(* CODESYS project aspersao_v1_1_0.library
   Company: Teknike
   DefaultNamespace: Teknike_Aspersao
   Version: 1.1.0
   Placeholder: Teknike_Aspersao
   Author: Tiago B. Cunico
   Description: Biblioteca para controle de aspersao
   Title: Aspersao

Project tree, tasks and I/O mapping:
  libraries: OSCAT - AixOCAT, * (RWTH Aachen University - E.ON Energy Research Center); Tc2_ControllerToolbox, * (Beckhoff Automation GmbH); Tc2_Standard, * (Beckhoff Automation GmbH); Tc2_System, * (Beckhoff Automation GmbH); Tc2_TcpIp, * (Beckhoff Automation GmbH); Tc2_Utilities, * (Beckhoff Automation GmbH); Tc3_Database, * (Beckhoff Automation GmbH); Tc3_Module, * (Beckhoff Automation GmbH); Geral, * (Teknike); Partidas, * (Teknike); Sensores, * (Teknike); SQL, * (Teknike); TwinCAT Dynamic String Kit, * (FisoThemes)
  POUs/
    Automatico/
      Aspercao/
        Balanca/
          function block FB_Balanca [ST]
          function block FB_SalvaBalancaBanco [ST]
          data type st_Balanca
        Camaras/
          Cluster/
            data type st_Cluster
            data type st_Cluster_Entrada
            data type st_Cluster_Interno
            data type st_Cluster_Saida
          function block FB_Camaras [ST]: AjustaSaidaPeV, AtualizaValvulasDosClusters, ContrlCamaras, ContrlCluster, ContrlEntreClusters, SalvaAbreEFechaNoCluster, DefineQuandoSalvaEvento, EventosRelatorio, fimAspersao, FimResfriamento, GeraRelatorio, InicioAspercao, InicioResfriamento, SalvaGrafico, SalvaProtocolo, AjustaEntrada, AjustaSaida, ControleLed, InicioPelaCamara, Status
          function block FB_SalvaEventoRelatorio [ST]: SalvaEvento
          data type st_Camara
          data type st_Camara_Config
          data type st_camara_Entradas
          data type st_camara_Saidas
          data type st_Camara_Status
          data type st_EventoRelatorio
        ControleLiberacaoCamaras/
          AreaFria/
            Sts/
              data type st_AreaFria
              data type st_AreaFriaControle
              data type st_SupervisorioAreaFria
            function block FB_ControleSaidaAreaFria [ST]: DefineQuandoSalvaEvento, EscrevePesoFrioCarcaca, EscrevePesoFrioProcesso, FimRefrimento, GeraRelatorio, IgnoraCarcacaBanco, SalvaEvento, AjustaEntrada, AjustaSaida, PegaCamarasDisponiveis, VeCarcacasAIgnorar
          AreaQuente/
            Sts/
              data type st_AreaQuente
              data type st_AreaQuenteControle
              data type st_SupCamarasDisponiveis
              data type st_SupervisorioAreaQuente
            function block FB_ControleEntradaAreaQuente [ST]: Cancela, EscreveNovaCarcacaBanco, EscreveNovoProcessoBanco, EscrevePesoQuenteProcesso, AjustaEntrada, AjustaSaida, PegaCamarasDisponiveis
          Funcionamento_TODO.txt
          data type st_CarcacaBD
          data type st_ProcessoBD
        ControleProtocolo/
          function block FB_ControleEdicaoProtocolo [ST]
          data type st_DBProtocolo
          data type st_Protocolo
        ControleValvulas/
          function block FB_ControleValvulaApersao [ST]: AjustaBanco, ControleEventos, EventosRelatorio, HoraTermina, LogBanco, SalvaAbreEFecha, AjustaEntrada, AjustaSaida, CancelaProtocolo, TempoMaximoDeProtocolo, VSAr
          data type st_ConfigControleValvula
          data type st_ControleValvula
          data type st_enControleValvulas
          data type st_saControleValvulas
          data type st_ValvulasBD
        RFIDeBalanca/
          function block FB_RFIDBalancaChoque [ST]: ControlePeso, ControleTAG
          function block FB_RFIDBalancaEntrada [ST]: ControlePeso, ControleTAG
          function block FB_RFIDBalancaSaida [ST]: ControlePeso, ControleTAG
          data type st_BufferTagBalanca
          data type st_RFIDdb
          data type st_RFIDePeso
      ControlesPID/
        Estruturas/
          data type stConfigMaxMinSet
          data type stControlePID
          data type stPID
          data type stPID_EN
          data type stPID_SA
        function block FB_PIDeGrafico [ST]: aPID, Grafico, TextoErro, TextoStatus
        data type st_Anel
        data type st_Tanque
    Comunicacao/
      sts/
        areafria/
          data type st_EnIHMAreaFria
          data type st_IHMAreaFria
          data type st_SaIHMAreaFria
        areaquente/
          data type st_EnIHMAreaQuente
          data type st_IHMAreaQuente
          data type st_SaIHMAreaQuente
        CamaraLRV/
          data type st_CamaraLRV
          data type st_En_CamaraLRV
          data type st_Sa_CamaraLRV
          data type st_StatusCamaras
        Camaras/
          data type st_En_IHMCamaras
          data type st_IHMCamara
          data type st_Sa_IHMCamaras
    global variables GVL_BlibliotecaAspersao
    program MAIN [ST]
    program ValidaLicensa [ST]: Licensas
  00000000-0000-0000-0000-000000000000|POUs\Automatico\Aspercao\ControleLiberacaoCamaras\Funcionamento_TODO.txt
*)

// POUs/Automatico/Aspercao/Balanca/st_Balanca
TYPE st_Balanca :
STRUCT
	xConecta : BOOL;	
	ip : T_IPv4Addr;
	xNovoResultado : BOOL;
	rPeso : REAL;
	xOnline : BOOL; //
	xResetContador : BOOL;
	iContador : UDINT;
	stBuffer : ARRAY[0..9] OF REAL;
END_STRUCT
END_TYPE

// POUs/Automatico/Aspercao/Camaras/Cluster/st_Cluster
TYPE st_Cluster :
STRUCT
	En 	: st_Cluster_Entrada;
	Sa 	: st_Cluster_Saida;
	i	: st_Cluster_Interno;
END_STRUCT
END_TYPE

// POUs/Automatico/Aspercao/Camaras/Cluster/st_Cluster_Entrada
TYPE st_Cluster_Entrada :
STRUCT
	iValvulas : ARRAY[0..20] OF INT;//Quais valvulas estao nesse cluster
	xPausaCluster : BOOL;//sinal da camara para sincronizar o cluster
	iPosisaoCluster : INT;//Em qual posição esse cluster esta, começa em 0
	rTempoEntreValvulas : REAL;//segundos entre cada 1 das valvulas
	xHabilitaEvaporador : ARRAY[0..10] OF BOOL;//Quais evaporadores vao parar quando esse cluster pedir
END_STRUCT
END_TYPE

// POUs/Automatico/Aspercao/Camaras/Cluster/st_Cluster_Interno
TYPE st_Cluster_Interno :
STRUCT
	
	
	rtMasterAbriu : R_TRIG;
	xHEaMestre : BOOL;
	dthrInicioValMestre : DT;//momento em que a valvula mestre inicio, usa pra saber quando libera o cluster
	xIniciaSincronismo : BOOL;// quando tru ele fica contando o tempo para quando for a hora liberar a valvula
	lrTempoTotal : LREAL;//essa é a divisao de quando cada valvula pode entrar, (tempo OFF mais Tempo ON)
	lrTempoDeCadaBloco : LREAL;//essa é a divisao de quando cada valvula pode entrar, (tempo OFF mais Tempo ON)/Numero de clusters
	lrPosicaoDeEntrada : LREAL;//momento em que a valvula pode entrar mesmo
	
	iEtapaAnterior : INT;
	
	rtIniciaSincronismo : R_TRIG;
	rtTrocouEtapa : R_TRIG;
	
	tonSincornismo : TON_P;
	TonMomentoDeEntrada : TON;
	rtMomentoDeEntrada : R_TRIG;
	
	btONOFFCluster : B_TRIG;
	
	tonCascata : TON;//controla a cascata de liga das valvulas
	xRodaCascata : BOOL;
	
	tonAjusteTempoCascata : TON;//Antes da cascata para conpensar as valvulas que ja abriram
	xAjustaCascata : BOOL;
	tTempoEsperaAntesCascata : TIME;
	
END_STRUCT
END_TYPE

// POUs/Automatico/Aspercao/Camaras/Cluster/st_Cluster_Saida
TYPE st_Cluster_Saida :
STRUCT
	iAbertas : INT;// quantas tao abertas agora
	xPausaValvula : ARRAY[0..20] OF BOOL;//Qual valvula tem que pausar
	iValvulaMestre : INT; //qual o index no array de valvulas que é a primeira valvula a ligar, usa essa como mestre das outras
	xLigadoAnterior : ARRAY[0..20] OF BOOL;//estado de qual esta ligada, quando uma muda de estado tem que fazer ela esperar ate sincronizar com a primeira
	
	xParaVentilacao : BOOL;//sinal para desligar a ventilação 
	
	xAlgumaValvulaAberta : BOOL;//OLha no cluster se tem alguma valvula aberta 
END_STRUCT
END_TYPE

// POUs/Automatico/Aspercao/Camaras/st_Camara
TYPE st_Camara :
STRUCT
	Config : st_Camara_Config;
	Status : st_Camara_Status;
	en	   : st_camara_Entradas;
	sa	   : st_camara_Saidas;
	Clusters : ARRAY[0..30] OF st_Cluster; // nao da pra ser maior que 50 
END_STRUCT
END_TYPE

// POUs/Automatico/Aspercao/Camaras/st_Camara_Config
TYPE st_Camara_Config :
STRUCT PERSISTENT
	sIPFTP : STRING;
	sAbreviacaoUnidade : STRING;
	xIgnoraBotaoFisico : BOOL;
	rTempoEsperaAntesAspergir : REAL;//conta esse tempo antes de começar o processo de aspersao
	
	rMaxTempCamara	: REAL;
	rMinTempCamara	: REAL;
	rMinUmidCamara	: REAL;
	rMaxUmidCamara	: REAL;
	
	sNome	: STRING;//nome da camara
	
	iTempoMaximoAspersao : UDINT;// Em horas
	iCarcacasAmostra : INT;
	iCarcacasReal : INT;
	
	
	iQuantidadeCamaras : INT := 3;//usadas para a conta
	iPosisaoCamara : INT; // posição em que a camara entra
	iOffSetCluster : INT; //se considera a mais ou a menos nos clusters da camara
	
	iCamara : INT;//numero da camara


	iValvulasAbertasNaCamara : INT;
	iMaxValvulasAbertasCamara : INT;


	xProtocoloPorCamara : BOOL;

	iSegDesligarVentilacao : INT;//tempo que vai segurar o sinal para desligar a ventilação antes e depois de ligar e desligar a valvula
	
	
	iProtocoloEscolhido : INT;

	stProtocolos: ARRAY[0..30] OF st_Protocolo;//Protolo dessa camara
	
	iIndexSensorTemperatura : INT;
	iIndexSensorUmidade : INT;
	
	xManualDesligaEvaporador : ARRAY[0..10] OF BOOL;//joga o sinal com a sala de maquinas para manual
	xSinalManualDesligaEvap : ARRAY[0..10] OF BOOL;//Aqui diz se é true ou false o sinal que vai pra la
	
	sValvulas : STRING;// valvula que estao nessa camara
	
	
	rTempoArAberto : REAL; //Tempo de ar aberto em segundos
	rTempoAntesDeAbrirOAr : REAL; //Tempo que ele espera antes de abrir a valvula de ar em segundos
	
END_STRUCT
END_TYPE

// POUs/Automatico/Aspercao/Camaras/st_camara_Entradas
TYPE st_camara_Entradas :
STRUCT
	rPressaoAnel 	: REAL;
	rTempTanque 	: REAL;
	rTempCamara		: REAL; //Temperatura da Camara
	rUmidadeCamara	: REAL; //Umidade da Camara


	xPausaUsuario 	: BOOL;
	
	sGuidAtual: STRING;// guid do processo que ela esta fazendo atualmente

	
	xFinalizaValvulasDaCamara : BOOL;
	xAtualizaValvulasCluster : BOOL;
	xHabilitaAtualizarCLuster : BOOL;
	
	xLigaTudoIHM : BOOL;
	xLigaTudoFisico : BOOL;
	xLigaTudoSupervisorio : BOOL;
	xIniciaCamaraIHM : BOOL;
	xFinalizaCamaraIHM : BOOL;
	xApagaProcessoSupervisorio : BOOL;
	xIniciaCamaraSupervisorio : BOOL;
	xFinalizaCamaraSupervisorio : BOOL;
	
	
	xLedManual : BOOL;
	xSinalManuLed : BOOL;	

	rPesosQuente : ARRAY[0..1000] OF REAL;
	rPesosFrio   : ARRAY[0..1000] OF REAL;
	
	stHoraAgora : TIMESTRUCT;
	
END_STRUCT
END_TYPE

// POUs/Automatico/Aspercao/Camaras/st_camara_Saidas
TYPE st_camara_Saidas :
STRUCT
	tHoraInicio 	: DT; //Hora de Inicio da Aspersão
	sHoraInicio 	: STRING; //q hrs vai terminar de aspergir a camara
	tHoraTermina	: DT; //Hora para o fim da Aspersão
	sHoraTermina 	: STRING; //q hrs vai terminar de aspergir a camara

	
	xLed : BOOL;
	
	iQuantidadeDeCluster : INT;// 
	
	iValvulas 			: ARRAY[0..30] OF INT;

	iValvulaMestraMestra : INT;//A valvula mestre mestre (braba dms)

	iStatusProcesso : INT;
	
	xDesligaEvaporador : ARRAY[0..10] OF BOOL;//Status de desligar calculado com base nos cluster
	
	lrTempoTotal : LREAL;//essa é a divisao de quando cada valvula pode entrar, (tempo OFF mais Tempo ON)
	lrTempoDeCadaBloco : LREAL;//essa é a divisao de quando cada valvula pode entrar, (tempo OFF mais Tempo ON)/Numero de clusters
	lrPosicaoDeEntrada : LREAL;//momento em que a valvula pode entrar mesmo
	xPodeIniciar : BOOL;//Sinal que a camara pode iniciar
	
END_STRUCT
END_TYPE

// POUs/Automatico/Aspercao/Camaras/st_Camara_Status
TYPE st_Camara_Status :
STRUCT
	sOndeFoiIniciado : STRING;
	xAlgumaValvulaEmManual : BOOL;
	xTodasValvulasCanceladas : BOOL;
	xPeloMenos1CanceladaOutrasAguradando : BOOL;
	xPegandoPesosQuentes : BOOL;
	xPegandoPesosFrios : BOOL;
	xTerminouAspercao: BOOL;//Status de que pode tirar as carcaças para testar o peso frio
	
	
	xCamaraTempOK	: BOOL; //Temperatura da camera esta OK
	xCamaraUmidOK	: BOOL; //Umidade da camera esta OK
	xAnelPressOK	: BOOL; //Pressao do anel esta OK
	xTanqueTempOK	: BOOL; //Temperatura do tanque esta OK
	
	
	iStatus			: INT; 
	sStatus : STRING;// status da camara
	
	
	sTempoAteCamaraEntrarNoSinc : STRING;
	sNomeProtocoloAtivo : STRING;//Nome do protocolo ativo

	iTagsAbreLiberacao : ARRAY[0..1] OF INT;
	iTagsFechaLiberacao : ARRAY[0..1] OF INT;
END_STRUCT
END_TYPE

// POUs/Automatico/Aspercao/Camaras/st_EventoRelatorio
TYPE st_EventoRelatorio :
STRUCT
	sGuid : STRING;
	xAtivo : BOOL;
	 
	iCamara : INT;
	Critico : BOOL;
	Tag : STRING;
	Descricao : STRING;
	Inicio : TIMESTRUCT;
	Fim : TIMESTRUCT;
END_STRUCT
END_TYPE

// POUs/Automatico/Aspercao/ControleLiberacaoCamaras/AreaFria/Sts/st_AreaFria
TYPE st_AreaFria :
STRUCT
	C : st_AreafriaControle;
	IHM : REFERENCE TO st_IHMAreaFria;
	Sup : st_SupervisorioAreaFria;
END_STRUCT
END_TYPE

// POUs/Automatico/Aspercao/ControleLiberacaoCamaras/AreaFria/Sts/st_AreaFriaControle
TYPE st_AreaFriaControle :
STRUCT
	iCamarasDisponiveis : ARRAY[0..50] OF INT; // para a lista do cara para escolher a camara
	iCamaraSelecionada	: INT;// qual camara o operador escolher para começar
	xIniciaCamara		: BOOL;// operador dizendo para começar a amostragem
	sGuidAtual			: STRING;// guid do processo atual
	
	xAleatorio			: BOOL;// se vai fazer a amostragem aleatorio ou sequencial
	sPesoBalanca		: STRING;//peso atual vindo da balança para o operador saber como que ta
	xCapturaPeso		: BOOL; // operador dizendo para pegar o peso atual
	
	rPesosQuentes		: ARRAY[0..20] OF REAL; // 	array com os pesos quentes amostrados pelo operador ou sequencialemnte
	rPesosFrios			: ARRAY[0..20] OF REAL; // 	array com os pesos frios amostrados pelo operador ou sequencialemnte
	
	rPesoAtual			: REAL;// Peso atual que vem da balança
	xPesoNovo			: BOOL;// Quando  balança diz que veio um peso novo
	
	
	iCarcacaAtual		: INT;// Qual o numero da carcaça que ele ta esperando
	
	xEmProcesso			: BOOL;
	
	xCancela 			: BOOL;

END_STRUCT
END_TYPE

// POUs/Automatico/Aspercao/ControleLiberacaoCamaras/AreaFria/Sts/st_SupervisorioAreaFria
TYPE st_SupervisorioAreaFria :
STRUCT
	
	stCamarasDisponiveis : ARRAY[0..50] OF st_SupCamarasDisponiveis;
	iCamaraSelecionada : INT;
	idSelecionadoCBCamara : INT;
	
	iModoDeAmostragem : INT;
	xIniciarAmostragem : BOOL;
	
	xCapturaAmostra : BOOL;
	xNovoPesoDebug : BOOL;
	rPesoDebug : REAL;
	
	
	iCarcacasAmostradas : INT;
	iCarcacasFaltaAmostrar : INT;
	iCarcacasAmostragemTotal : INT;
	
	
END_STRUCT
END_TYPE

// POUs/Automatico/Aspercao/ControleLiberacaoCamaras/AreaQuente/Sts/st_AreaQuente
TYPE st_AreaQuente :
STRUCT
	C : st_AreaQuenteControle;
	IHM : REFERENCE TO st_IHMAreaQuente;
	Sup : st_SupervisorioAreaQuente;
END_STRUCT
END_TYPE

// POUs/Automatico/Aspercao/ControleLiberacaoCamaras/AreaQuente/Sts/st_AreaQuenteControle
TYPE st_AreaQuenteControle :
STRUCT
	iCamarasDisponiveis : ARRAY[0..50] OF INT; // para a lista do cara para escolher a camara
	iCamaraSelecionada	: INT;// qual camara o operador escolher para começar
	xIniciaCamara		: BOOL;// operador dizendo para começar a amostragem
	sGuidAtual			: STRING;// guid do processo atual
	
	xAleatorio			: BOOL;// se vai fazer a amostragem aleatorio ou sequencial
	sPesoBalanca		: STRING;//peso atual vindo da balança para o operador saber como que ta
	xCapturaPeso		: BOOL; // operador dizendo para pegar o peso atual
	
	rPesosQuentes		: ARRAY[0..20] OF REAL; // 	array com os pesos quentes amostrados pelo operador ou sequencialemnte
	rPesosFrio			: ARRAY[0..20] OF REAL; // 	array com os pesos quentes amostrados pelo operador ou sequencialemnte
	
	rPesoAtual			: REAL;// Peso atual que vem da balança
	xPesoNovo			: BOOL;// Quando  balança diz que veio um peso novo
	
	iCarcacaAtual		: INT;// Qual o numero da carcaça que ele ta esperando
	
	xEmProcesso			: BOOL;
	
	xCancela 			: BOOL;
	
	xPesoColetadoRX		: BOOL;
	
	
END_STRUCT
END_TYPE

// POUs/Automatico/Aspercao/ControleLiberacaoCamaras/AreaQuente/Sts/st_SupCamarasDisponiveis
TYPE st_SupCamarasDisponiveis :
STRUCT
	sNome : STRING;
	iCamara : INT;
END_STRUCT
END_TYPE

// POUs/Automatico/Aspercao/ControleLiberacaoCamaras/AreaQuente/Sts/st_SupervisorioAreaQuente
TYPE st_SupervisorioAreaQuente :
STRUCT
	stCamarasDisponiveis : ARRAY[0..50] OF st_SupCamarasDisponiveis;
	iCamaraSelecionada : INT;
	idSelecionadoCBCamara : INT;
	
	iModoDeAmostragem : INT;
	xIniciarAmostragem : BOOL;
	
	xCapturaAmostra : BOOL;
	xNovoPesoDebug : BOOL;
	rPesoDebug : REAL;
	
	
	iCarcacasAmostradas : INT;
	iCarcacasFaltaAmostrar : INT;
	iCarcacasAmostragemTotal : INT;
	
	
END_STRUCT
END_TYPE

// POUs/Automatico/Aspercao/ControleLiberacaoCamaras/st_CarcacaBD
TYPE st_CarcacaBD :
STRUCT
	ID: DINT;
	Camara: DINT;
	Processo: STRING(40);
	nCarcaca: DINT;
	PesoQuente: LREAL;
	horaPesoQuente: DT;
	PesoFrio: LREAL;
	horaPesoFrio: DT;
	Status: STRING(45);
	Timestamp: DT;
END_STRUCT
END_TYPE

// POUs/Automatico/Aspercao/ControleLiberacaoCamaras/st_ProcessoBD
TYPE st_ProcessoBD :
STRUCT
	Processo: STRING(40);
	Camara: DINT;
	InicioResfriamento: DT;
	FimResfriamento: DT;
	InicioAspersao: DT;
	FimAspersao: DT;
	NumeroCarcacas: DINT;
	ConsumoAguaTotal: LREAL;
	Cancelado: SINT;
	Finalizado: SINT;
	Aspergida: SINT;
	Pesoquente: LREAL;
	PesoFrio: LREAL;
	Status: STRING(45);
	Timestamp: DT;
END_STRUCT
END_TYPE

// POUs/Automatico/Aspercao/ControleProtocolo/st_DBProtocolo
TYPE st_DBProtocolo :
STRUCT RETAIN PERSISTENT
	ID: DINT;
	Nome: STRING(100);
	NomeIHM: STRING(20);
	Valvulas: STRING(255);
	ET01TON: LREAL;
	ET01TOFF: LREAL;
	ET01NC: DINT;
	ET02TON: LREAL;
	ET02TOFF: LREAL;
	ET02NC: DINT;
	ET03TON: LREAL;
	ET03TOFF: LREAL;
	ET03NC: DINT;
	ET04TON: LREAL;
	ET04TOFF: LREAL;
	ET04NC: DINT;
	ET05TON: LREAL;
	ET05TOFF: LREAL;
	ET05NC: DINT;
	ET06TON: LREAL;
	ET06TOFF: LREAL;
	ET06NC: DINT;
	ET07TON: LREAL;
	ET07TOFF: LREAL;
	ET07NC: DINT;
	ET08TON: LREAL;
	ET08TOFF: LREAL;
	ET08NC: DINT;
	ET09TON: LREAL;
	ET09TOFF: LREAL;
	ET09NC: DINT;
	ET10TON: LREAL;
	ET10TOFF: LREAL;
	ET10NC: DINT;
END_STRUCT
END_TYPE

// POUs/Automatico/Aspercao/ControleProtocolo/st_Protocolo
TYPE st_Protocolo :
STRUCT
	xEditado : BOOL;
	xSelecionado : BOOL;
	DB : st_DBProtocolo;
END_STRUCT
END_TYPE

// POUs/Automatico/Aspercao/ControleValvulas/st_ConfigControleValvula
TYPE st_ConfigControleValvula :
STRUCT PERSISTENT
	sNomeValvulaIHM : STRING;
	rTempoArAberto : REAL; //Tempo de ar aberto em segundos
	rTempoAntesDeAbrirOAr : REAL; //Tempo que ele espera antes de abrir a valvula de ar em segundos
END_STRUCT
END_TYPE

// POUs/Automatico/Aspercao/ControleValvulas/st_ControleValvula
TYPE st_ControleValvula :
STRUCT 
	EN	: st_enControleValvulas;
	SA	: st_saControleValvulas;
	Config : st_ConfigControleValvula;
	//DB 	: st_ValvulasBD;//st do banco
	
END_STRUCT
END_TYPE

// POUs/Automatico/Aspercao/ControleValvulas/st_enControleValvulas
TYPE st_enControleValvulas :
STRUCT
	stValvula 		: REFERENCE TO st_Valvula;//Estrutura da valvula que vai ser controlada
	iIndexValvula 	: INT; //index da valvula que é controlada

	stValvulaAR 	: REFERENCE TO st_Valvula;//Estrutura da valvula que vai ser controlada
	iIndexValvulaAR	: INT; //index da valvula que é controlada
	
	sIHM 			: ARRAY[0..4] OF STRING;//textos que vao pra IHM
	stProtocolos 	: ARRAY[0..4] OF st_Protocolo;// Protocolos que podem ser usados nesta valvula
	stProtoEscolhido: st_Protocolo;
	
	GUID			: STRING;//GUID do processo que vai ser feito na valvula, se for 0 é pq nao tem proceso rolando, ai nao pode aspergir
	xCamaraTempOK	: BOOL; //Temperatura da camera esta OK
	xCamaraUmidOK	: BOOL; //Umidade da camera esta OK
	xAnelPressOK	: BOOL; //Pressao do anel esta OK
	xTanqueTempOK	: BOOL; //Temperatura do tanque esta OK
	
	xBloqueado		: BOOL;	//Nao pode iniciar o processo por falta de alguma coisa, pode ser que nao foi iniciado o processo ou que nao pode iniciar a asperção
	
	rTempAgua		: REAL; //temperatura da agua para o log no banco
	rPressaoAnel	: REAL;	//pressao da anel para o log no banco
	tsHoraAtual		: TIMESTRUCT; //Hora atual
	
	xCancela		: BOOL; //sinal de cancela o protocolo atual
	
	iMaxValvulas	: INT; //Quantidade maxima de valvulas abertas
	iValvulasAbertas: REFERENCE TO INT; //Quantidade de valvulas abetas no momento
	iValvulasAbertasCamara : REFERENCE TO INT;
	iMaxValvulasAbertasCamara : INT;
	
	xPulaAspersao 	: BOOL;//vai para o fim da aspersao como se tivesse tudo certo
	
	xLigaManual : BOOL;//liga em manual e gera o evento no relatorio
	
	xFinalizaInterno : BOOL;// finaliza a aspersao da valvula, a principio é so interno
	
	iCluster : INT;// o cluster que foi escolhido para essa valvula
	
	xPausaSincCluster : BOOL;//pausa para o sincronismo das valvulas do cluster
	xPausaSincEntreCluster : BOOL;//pausa para o sincronismo entre clusters
	xPausaSincCamaras : BOOL;//pausa para o sincronismo entre as camaras
	
	iTempoMaximoAspersao : UDINT;// Em horas que pode ficar fazendo a aspersao
	
	iSegDesligarVentilacao : INT;//tempo que vai segurar o sinal para desligar a ventilação antes e depois de ligar e desligar a valvula
	
	sNomeCamara : STRING;
	
	xLigaAutomaticoSupervisorio : BOOL;
	xLigaManualSupervisorio : BOOL;
	xCancelaSupervisorio : BOOL;
	
	tTempoAteSinc : TIME;//Tempo ate a valvula sincronizar
	
	rTempoEsperaAntesAspergir : REAL;//conta esse tempo antes de começar o processo de aspersao
	
	
	xLigaManualARSupervisorio : BOOL;
	
END_STRUCT
END_TYPE

// POUs/Automatico/Aspercao/ControleValvulas/st_saControleValvulas
TYPE st_saControleValvulas :
STRUCT
	iStatus : INT;
	sStatus : STRING;
	xEmProcesso : BOOL;// se a valvula ja escolheu o protocolo e vai tentar aspergir
	xValvulaAberta : BOOL;
	xPausado: BOOL;
	xFinalizou : BOOL;
	sTempoRestante : STRING(16);
	sCiclo: STRING(6);
	
	dtHoraInicio : DT;// que hrs inicio o protocolo
	sHoraInicio : STRING;//que hrs inicio o protocolo
	dtHoraTermina : DT;// que hrs termina o protocolo
	sHoraTermina : STRING;//que hrs termina o protocolo
	
	iTotalDeCiclos : INT;// quantidade de ciclos que o protocolo tem
	rEtapasSemMudar: ARRAY[1..10,1..3] OF LREAL;//etapas do processo sem alterar durante o processo
	iEtapaAtual : INT;//Etapa atual do processo
	xNaoLigoSoPorSincETC : BOOL; //sinal de que so nao liga por sincronismo entre clusters
	xPausadoSemSin : BOOL; //sinal de que pausou por alguma coisa que nao é sincronismo
	xParaVentilacao : BOOL;//sinal para desligar a ventilação 
	sNomeProtocoloAtivo : STRING;//Nome do protocolo ativo
	
	sStatusAr : STRING;
	xMandaArAbrir : BOOL;
	iStatusVsAr : INT;
END_STRUCT
END_TYPE

// POUs/Automatico/Aspercao/ControleValvulas/st_ValvulasBD
TYPE st_ValvulasBD :
STRUCT RETAIN PERSISTENT
	ID: DINT;
	Valvula: DINT;
	Processo: STRING(40);
	protocolo: DINT;
	Ciclo: DINT;
	Inicio: DT;
	Fim: DT;
	Aspergindo: DT;
	NaoAspergindo: DT;
	Pausado: DT;
	vazao: LREAL;
	TemperaturaAgua: LREAL;
	PressaoAnel: LREAL;
	Cancelado: SINT;
	Timestamp: DT;
END_STRUCT
END_TYPE

// POUs/Automatico/Aspercao/RFIDeBalanca/st_BufferTagBalanca
TYPE st_BufferTagBalanca :
STRUCT
	iTag : INT;
	rPeso : REAL;
END_STRUCT
END_TYPE

// POUs/Automatico/Aspercao/RFIDeBalanca/st_RFIDdb
TYPE st_RFIDdb :
STRUCT
	ID: DINT;
	TAG: STRING(45);
	Processo: STRING(40);
	Camara: DINT;
	Trilho: STRING(45);
	Trecho: STRING(45);
	nCarcaca: DINT;
	PesoQuente: LREAL;
	HoraPesoQuente: DT;
	PesoFrio: LREAL;
	HoraPesoFrio: DT;
	status: STRING(100);
	Protocolo: STRING(45);
	InicioProtocolo: DT;
	FimProtocolo: DT;
END_STRUCT
END_TYPE

// POUs/Automatico/Aspercao/RFIDeBalanca/st_RFIDePeso
TYPE st_RFIDePeso :
STRUCT
	
	xLimpaFilaPeso : BOOL;
	xLimpaFilaTAG : BOOL;
	
	
	stBuffer : ARRAY[0..9] OF st_BufferTagBalanca;
END_STRUCT
END_TYPE

// POUs/Automatico/ControlesPID/Estruturas/stConfigMaxMinSet
TYPE stConfigMaxMinSet :
STRUCT RETAIN PERSISTENT
	rSetpoint : REAL;
	rMax : REAL;
	rMin : REAL;
END_STRUCT
END_TYPE

// POUs/Automatico/ControlesPID/Estruturas/stControlePID
TYPE stControlePID :
STRUCT
	Config : stConfigMaxMinSet;
	PID : stPID;
	Grafico : ARRAY[0..3,0..120] OF ST_Grafico;//amostragem a cada 0.5 s. Pressao atual, setpoint, saida do PID?
	xLigaSistema : BOOL;
	xLigaInterno : BOOL;
	xModoCalibracao : BOOL;
	rOutraNoGrafico : REAL;
	xPressao : BOOL;
	xReset : BOOL;
END_STRUCT
END_TYPE

// POUs/Automatico/ControlesPID/Estruturas/stPID
TYPE stPID :
STRUCT RETAIN PERSISTENT
	EN : stPID_EN;
	SA : stPID_SA;
	stParams : ST_CTRL_PID_PARAMS;
END_STRUCT
END_TYPE

// POUs/Automatico/ControlesPID/Estruturas/stPID_EN
TYPE stPID_EN :
STRUCT
	fSetpointValue    : FLOAT;
    fActualValue      : FLOAT;
    fManSyncValue     : FLOAT;
    bSync             : BOOL;
    eMode             : E_CTRL_MODE;
    bHold             : BOOL;
	rMaximo			  : REAL;
	rMinimo			  : REAL;
END_STRUCT
END_TYPE

// POUs/Automatico/ControlesPID/Estruturas/stPID_SA
TYPE stPID_SA :
STRUCT
	fOut          : FLOAT;
    bARWactive    : BOOL;
    eState        : E_CTRL_STATE;
    sState        : STRING;
    eErrorId      : E_CTRL_ERRORCODES;
    sErrorId      : STRING;
    bError        : BOOL;
	rSaida		  : REAL;
END_STRUCT
END_TYPE

// POUs/Automatico/ControlesPID/st_Anel
TYPE st_Anel :
STRUCT
	xPressaoOK : BOOL;
	rPressaoInicio : REAL;
	rPressaoFim : REAL;
	rTempInicio : REAL;
	rTempFim : REAL;
	rPorcetagemValvula : REAL;
END_STRUCT
END_TYPE

// POUs/Automatico/ControlesPID/st_Tanque
TYPE st_Tanque :
STRUCT
	xTempOk : BOOL;
	rTempSaida : REAL;
	rTempTrocador : REAL;
	rNivelQuente : REAL;
	rNivelFrio : REAL;
END_STRUCT
END_TYPE

// POUs/Comunicacao/sts/areafria/st_EnIHMAreaFria
TYPE st_EnIHMAreaFria :
STRUCT
	
	iCamaraLiberacaoTX AT %I* : INT;
	xColetaAmostraX AT %I* : BOOL;
	xFinalizaCarregamentoTX AT %I* : BOOL;
	xColocaCamaraStandbyTX AT %I* : BOOL;
	xConsecutivoTX AT %I* : BOOL;
	xAleatorioTX AT %I* : BOOL;
	xAutomaticoTX AT %I* : BOOL;
	xIniciaAmostragemSequencialTX AT %I* : BOOL;
	xIniciaCamaraTX AT %I* : BOOL;
	xCancelaAmostragemTX AT %I* : BOOL;
	xConfirmaFinalAmostragem AT %I* : BOOL;
	
	xIgnoraCarcaca AT %I* : ARRAY[0..20] OF BOOL;


END_STRUCT
END_TYPE

// POUs/Comunicacao/sts/areafria/st_IHMAreaFria
TYPE st_IHMAreaFria :
STRUCT
	EN : st_EnIHMAreaFria;
	SA : st_SAIHMAreafria;
END_STRUCT
END_TYPE

// POUs/Comunicacao/sts/areafria/st_SaIHMAreaFria
TYPE st_SaIHMAreaFria :
STRUCT
	
	rPesoFrioAtualRX AT %Q* : REAL;
	iAmostraAtualRX AT %Q* : INT;
	iFaltaAmostrarRX AT %Q* : INT;
	iQtdAmostradaRX AT %Q* : INT;
	iTagRFIDRX AT %Q* : INT;
	iCamaraCarregementoTX AT %Q* : INT;
	xFinalizouAmostragrmRX AT %Q* : BOOL;
	xCamaraSelecionadaLiberadaRX AT %Q* : BOOL;
	xSistemaLiberadoParaIniciar AT %Q* : BOOL;
	xEmProcesso AT %Q* : BOOL;
	xPesoColetadoRX AT %Q* : BOOL;
	iPercentualAmostrado AT %Q* : INT;
	
	iTempoFinalResfriamento AT %Q* : 	INT;
	rTempoFinalResfriamento AT %Q* : 	REAL;
	
	sStatus1 AT %Q* : STRING(25);
	sStatus2 AT %Q* : STRING(25);
	sStatus3 AT %Q* : STRING(25);
	sStatus4 AT %Q* : STRING(25);
	sStatus5 AT %Q* : STRING(25);
	sStatus6 AT %Q* : STRING(25);
	sStatus7 AT %Q* : STRING(25);
	sStatus8 AT %Q* : STRING(25);
	sStatus9 AT %Q* : STRING(25);
	sStatus10 AT %Q* : STRING(25);
	rTempCam1 AT %Q* : REAL;
	rTempCam2 AT %Q* : REAL;
	rTempCam3 AT %Q* : REAL;
	rTempCam4 AT %Q* : REAL;
	rTempCam5 AT %Q* : REAL;
	rTempCam6 AT %Q* : REAL;
	rTempCam7 AT %Q* : REAL;
	rTempCam81 AT %Q* : REAL;
	rTempCam82 AT %Q* : REAL;
	rTempCam9 AT %Q* : REAL;
	
	
	iCarcacaIgnorada AT %Q* : ARRAY[0..20] OF INT;
	sPesoCaraca AT %Q* : ARRAY[0..20] OF STRING(25);


END_STRUCT
END_TYPE

// POUs/Comunicacao/sts/areaquente/st_EnIHMAreaQuente
TYPE st_EnIHMAreaQuente :
STRUCT
	
	iCamaraCarregementoTX AT %I* : INT;
	xColetaAmostraTX AT %I* : BOOL;
	xFinalizaCarregamentoTX AT %I* : BOOL;
	xColocaCamaraStandbyTX AT %I* : BOOL;
	xConsecutivoAqTX AT %I* : BOOL;
	xAleatorioAqTX AT %I* : BOOL;
	xAutomaticoAQTX AT %I* : BOOL;
	xIniciaAmostragemSequencialTX AT %I* : BOOL;
	xIniciaCamaraTX AT %I* : BOOL;
	xCancelaAmostragemTX AT %I* : BOOL;
	xConfirmaFinalAmostragem AT %I* : BOOL;


END_STRUCT
END_TYPE

// POUs/Comunicacao/sts/areaquente/st_IHMAreaQuente
TYPE st_IHMAreaQuente :
STRUCT
	EN : st_EnIHMAreaQuente;
	SA : st_SAIHMAreaQuente;
END_STRUCT
END_TYPE

// POUs/Comunicacao/sts/areaquente/st_SaIHMAreaQuente
TYPE st_SaIHMAreaQuente :
STRUCT
	
	rPesoQuenteAtualRX AT %Q* : REAL;
	iAmostraAtualRX AT %Q* : INT;
	iFaltaAmostrarRX AT %Q* : INT;
	iQtdAmostradaRX AT %Q* : INT;
	iTagRFIDRX AT %Q* : INT;
	iCamaraCarregementoTX AT %Q* : INT;
	xFinalizouAmostragrmRX AT %Q* : BOOL;
	xCamaraSelecionadaLiberadaRX AT %Q* : BOOL;
	xSistemaLiberadoParaIniciar AT %Q* : BOOL;
	xEmProcesso AT %Q* : BOOL;
	xPesoColetadoRX AT %Q* : BOOL;
	iPercentualAmostrado AT %Q* : INT;
	sStatus1 AT %Q* : STRING(25);
	sStatus2 AT %Q* : STRING(25);
	sStatus3 AT %Q* : STRING(25);
	sStatus4 AT %Q* : STRING(25);
	sStatus5 AT %Q* : STRING(25);
	sStatus6 AT %Q* : STRING(25);
	sStatus7 AT %Q* : STRING(25);
	sStatus8 AT %Q* : STRING(25);
	sStatus9 AT %Q* : STRING(25);
	sStatus10 AT %Q* : STRING(25);


END_STRUCT
END_TYPE

// POUs/Comunicacao/sts/CamaraLRV/st_CamaraLRV
TYPE st_CamaraLRV :
STRUCT
	En : st_En_CamaraLRV;
	Sa : st_Sa_CamaraLRV;
END_STRUCT
END_TYPE

// POUs/Comunicacao/sts/CamaraLRV/st_En_CamaraLRV
TYPE st_En_CamaraLRV :
STRUCT
	
	iCamaraSelecionada AT %I* : INT;
	iProtocoloSelecionado AT %I* : INT;
	xLigaValvulaC1_1 AT %I* : BOOL;
	xLigaValvulaC1_2 AT %I* : BOOL;
	xLigaValvulaC1_3 AT %I* : BOOL;
	xLigaValvulaC1_4 AT %I* : BOOL;
	xLigaValvulaC1_5 AT %I* : BOOL;
	xLigaValvulaC1_6 AT %I* : BOOL;
	xLigaValvulaC1_7 AT %I* : BOOL;
	xLigaValvulaC1_8 AT %I* : BOOL;
	xLigaValvulaC1_9 AT %I* : BOOL;
	xLigaValvulaC1_10 AT %I* : BOOL;
	xLigaValvulaC1_11 AT %I* : BOOL;
	xLigaValvulaC1_12 AT %I* : BOOL;
	xLigaValvulaC1_13 AT %I* : BOOL;
	xCancelaC1_1 AT %I* : BOOL;
	xCancelaC1_2 AT %I* : BOOL;
	xCancelaC1_3 AT %I* : BOOL;
	xCancelaC1_4 AT %I* : BOOL;
	xCancelaC1_5 AT %I* : BOOL;
	xCancelaC1_6 AT %I* : BOOL;
	xCancelaC1_7 AT %I* : BOOL;
	xCancelaC1_8 AT %I* : BOOL;
	xCancelaC1_9 AT %I* : BOOL;
	xCancelaC1_10 AT %I* : BOOL;
	xCancelaC1_11 AT %I* : BOOL;
	xCancelaC1_12 AT %I* : BOOL;
	xCancelaC1_13 AT %I* : BOOL;
	xLigaManualC1_1 AT %I* : BOOL;
	xLigaManualC1_2 AT %I* : BOOL;
	xLigaManualC1_3 AT %I* : BOOL;
	xLigaManualC1_4 AT %I* : BOOL;
	xLigaManualC1_5 AT %I* : BOOL;
	xLigaManualC1_6 AT %I* : BOOL;
	xLigaManualC1_7 AT %I* : BOOL;
	xLigaManualC1_8 AT %I* : BOOL;
	xLigaManualC1_9 AT %I* : BOOL;
	xLigaManualC1_10 AT %I* : BOOL;
	xLigaManualC1_11 AT %I* : BOOL;
	xLigaManualC1_12 AT %I* : BOOL;
	xLigaManualC1_13 AT %I* : BOOL;
	xIniciaAspersaoC1 AT %I* : BOOL;
	xFinalizaAspersaoC1 AT %I* : BOOL;

END_STRUCT
END_TYPE

// POUs/Comunicacao/sts/CamaraLRV/st_Sa_CamaraLRV
TYPE st_Sa_CamaraLRV :
STRUCT
	
	sTempoC1_1 AT %Q* : STRING(16);
	sTempoC1_2 AT %Q* : STRING(16);
	sTempoC1_3 AT %Q* : STRING(16);
	sTempoC1_4 AT %Q* : STRING(16);
	sTempoC1_5 AT %Q* : STRING(16);
	sTempoC1_6 AT %Q* : STRING(16);
	sTempoC1_7 AT %Q* : STRING(16);
	sTempoC1_8 AT %Q* : STRING(16);
	sTempoC1_9 AT %Q* : STRING(16);
	sTempoC1_10 AT %Q* : STRING(16);
	sTempoC1_11 AT %Q* : STRING(16);
	sTempoC1_12 AT %Q* : STRING(16);
	sTempoC1_13 AT %Q* : STRING(16);
	sTempoC1_14 AT %Q* : STRING(16);
	sTempoC1_15 AT %Q* : STRING(16);
	sTempoC1_16 AT %Q* : STRING(16);
	sTempoC1_17 AT %Q* : STRING(16);
	sTempoC1_18 AT %Q* : STRING(16);
	sTempoC1_19 AT %Q* : STRING(16);
	sTempoC1_20 AT %Q* : STRING(16);
	sTempoC1_21 AT %Q* : STRING(16);
	sTempoC1_22 AT %Q* : STRING(16);
	sTempoC1_23 AT %Q* : STRING(16);
	sTempoC1_24 AT %Q* : STRING(16);
	sTempoC1_25 AT %Q* : STRING(16);
	sTempoC1_26 AT %Q* : STRING(16);
	iStatusC1_1 AT %Q* : INT;
	iStatusC1_2 AT %Q* : INT;
	iStatusC1_3 AT %Q* : INT;
	iStatusC1_4 AT %Q* : INT;
	iStatusC1_5 AT %Q* : INT;
	iStatusC1_6 AT %Q* : INT;
	iStatusC1_7 AT %Q* : INT;
	iStatusC1_8 AT %Q* : INT;
	iStatusC1_9 AT %Q* : INT;
	iStatusC1_10 AT %Q* : INT;
	iStatusC1_11 AT %Q* : INT;
	iStatusC1_12 AT %Q* : INT;
	iStatusC1_13 AT %Q* : INT;
	iStatusC1_14 AT %Q* : INT;
	iStatusC1_15 AT %Q* : INT;
	iStatusC1_16 AT %Q* : INT;
	iStatusC1_17 AT %Q* : INT;
	iStatusC1_18 AT %Q* : INT;
	iStatusC1_19 AT %Q* : INT;
	iStatusC1_20 AT %Q* : INT;
	iStatusC1_21 AT %Q* : INT;
	iStatusC1_22 AT %Q* : INT;
	iStatusC1_23 AT %Q* : INT;
	iStatusC1_24 AT %Q* : INT;
	iStatusC1_25 AT %Q* : INT;
	iStatusC1_26 AT %Q* : INT;
	xEmprocessoC1 AT %Q* : BOOL;
	
	sCicloC1_V1 AT %Q* : STRING(6);
	sCicloC1_V2 AT %Q* : STRING(6);
	sCicloC1_V3 AT %Q* : STRING(6);
	sCicloC1_V4 AT %Q* : STRING(6);
	sCicloC1_V5 AT %Q* : STRING(6);
	sCicloC1_V6 AT %Q* : STRING(6);
	sCicloC1_V7 AT %Q* : STRING(6);
	sCicloC1_V8 AT %Q* : STRING(6);
	sCicloC1_V9 AT %Q* : STRING(6);
	sCicloC1_V10 AT %Q* : STRING(6);
	sCicloC1_V11 AT %Q* : STRING(6);
	sCicloC1_V12 AT %Q* : STRING(6);
	sCicloC1_V13 AT %Q* : STRING(6);
	sCicloC1_V14 AT %Q* : STRING(6);
	sCicloC1_V15 AT %Q* : STRING(6);
	sCicloC1_V16 AT %Q* : STRING(6);
	sCicloC1_V17 AT %Q* : STRING(6);
	sCicloC1_V18 AT %Q* : STRING(6);
	sCicloC1_V19 AT %Q* : STRING(6);
	sCicloC1_V20 AT %Q* : STRING(6);
	sCicloC1_V21 AT %Q* : STRING(6);
	sCicloC1_V22 AT %Q* : STRING(6);
	sCicloC1_V23 AT %Q* : STRING(6);
	sCicloC1_V24 AT %Q* : STRING(6);
	sCicloC1_V25 AT %Q* : STRING(6);
	sCicloC1_V26 AT %Q* : STRING(6);



END_STRUCT
END_TYPE

// POUs/Comunicacao/sts/CamaraLRV/st_StatusCamaras
TYPE st_StatusCamaras :
STRUCT
	wReservasRX AT %I* : ARRAY[1..10] OF WORD;
	wReservasTX AT %Q* : ARRAY[1..10] OF WORD;
	
	sStatusDireita AT %Q* : STRING(25);
	sStatusEsquerda AT %Q* : STRING(25);
	sStatusDireitaBaixo AT %Q* : STRING(25);
	sStatusEsquerdaBaixo AT %Q* : STRING(25);
	sStatusInferiorBaixo AT %Q* : STRING(25);
	sStatusInferiorMeio AT %Q* : STRING(25);
	sStatusInferiorAlto AT %Q* : STRING(25);
	sStatusReserva6 AT %Q* : STRING(25);
	sStatusReserva7 AT %Q* : STRING(25);
	sStatusReserva8 AT %Q* : STRING(25);
	sStatusReserva9 AT %Q* : STRING(25);
	sStatusReserva10 AT %Q* : STRING(25);
END_STRUCT
END_TYPE

// POUs/Comunicacao/sts/Camaras/st_En_IHMCamaras
TYPE st_En_IHMCamaras :
STRUCT
	iCamaraValvula AT %I* : INT;
	xInverte1VS AT %I* : BOOL;
	xInverte2VS AT %I* : BOOL;
	xInverte3VS AT %I* : BOOL;
	iProtocoloSelecionado AT %I* : INT;
	xLigaCamara AT %I* : BOOL;
	xCancelaCamara AT %I* : BOOL;
	xPausaCamara AT %I* : BOOL;
END_STRUCT
END_TYPE

// POUs/Comunicacao/sts/Camaras/st_IHMCamara
TYPE st_IHMCamara :
STRUCT
	En : st_En_IHMCamaras;
	Sa : st_Sa_IHMCamaras;
END_STRUCT
END_TYPE

// POUs/Comunicacao/sts/Camaras/st_Sa_IHMCamaras
TYPE st_Sa_IHMCamaras :
STRUCT
	sTempoV1 AT %Q* : STRING(254);
	sTempoV2 AT %Q* : STRING(254);
	sTempoV3 AT %Q* : STRING(20);
	
	xLiberadoParaAspersao AT %Q* : BOOL;
	iValvulasAbertasAnel1 AT %Q* : INT;
	iValvulasAbertasAnel2 AT %Q* : INT;
	iValvulasAbertasAnel3 AT %Q* : INT;
	rNivelReservatorio AT %Q* : REAL;	
	
	iStatus1Valvula AT %Q* : INT;
	iStatus2Valvula AT %Q* : INT;
	iStatus3Valvula AT %Q* : INT;
END_STRUCT
END_TYPE

// POUs/GVL_BlibliotecaAspersao
//{attribute 'qualified_only'}
VAR_GLOBAL
    {attribute 'hide'} 
	{attribute 'tc_no_symbol'}
	xLicensaValida6446896834 : BOOL;
	LicensaValida : BOOL;
	STCheckLicense : ST_CheckLicense;
END_VAR

// POUs/Automatico/Aspercao/Balanca/FB_Balanca
//{attribute 'hide_all_locals'}
FUNCTION_BLOCK FB_Balanca
VAR_INPUT
	xConecta : BOOL := false;	
	ip : T_IPv4Addr := '192.168.100.20';
	xTipo : INT;//tipo da balanca 0 = marel, 1 = lenk
	xResetCOntador : BOOL;
END_VAR
VAR_OUTPUT
	xNovoResultado : BOOL;
	xOnline : BOOL; //
	rPeso : REAL;
	iContador : UDINT;
	stBuffer : ARRAY[0..9] OF REAL;
END_VAR
VAR	
	xAmostra : BOOL;

	fbConection : FB_ClientServerConnection;
	fbRecebe : FB_SocketReceive;
	sRecebido: STRING(1000);
	sRecebidoB: STRING(1000);
	rtTerminouDeMandarOComando : R_TRIG;
	tPeraUmPoucoAntesDePedirOqueVeio : TON;
	xManda: BOOL;
	tEspera : TIME;
	rtAmostra : R_TRIG;
	sAjustado: STRING(1000);
	
	
	iPos : DINT;
	

	iaux : INT;

	//fba : FB_StringBuilder;
	raux : REAL;
	
	
	
	i : INT;
	
	
	nErrId : UDINT;
	
	tofOffline : TOF;
	
	xAuxOnline : BOOL;
	
	tonPodeReceberLeitura : TON;
	
	sTeste : STRING;
	
	iDelete : INT := 9;
	iLeft	: INT := 5;
	
END_VAR

IF TRUE THEN	
	

	CASE xTipo OF
		
		0://marel
			xNovoResultado := FALSE;
			
			//Auto reset na conexao
			tonPodeReceberLeitura(IN:= TRUE, PT:= T#30M, Q=> , ET=> );
			IF tonPodeReceberLeitura.q THEN
				tonPodeReceberLeitura(IN:= FALSE);
				fbConection(bEnable:= FALSE);
			END_IF
			
			
			//conecta na tcp socket
			fbConection(
				sSrvNetID:= '', 
				nMode:= CONNECT_MODE_ENABLEDBG, 
				sRemoteHost:= ip, 
				nRemotePort:= 52211, 
				bEnable:= xConecta, 
				tReconnect:= T#1S, 
				bBusy=> , 
				bError=> , 
				nErrId=> , 
				hSocket=> , 
				eState=> );
				
				
			IF NOT fbConection.bBusy THEN
				xAuxOnline := xConecta;
				IF fbConection.bError THEN
					nErrId := fbConection.nErrId;
					xAuxOnline := FALSE;
				END_IF
			END_IF
			
			tofOffline(IN:= xAuxOnline, PT:= T#5S, Q=> xOnline, ET=> );
				
			
			//fica rodando o recebe pra ficar lendo caso aparece alguma coisa
			IF NOT fbRecebe.bExecute THEN
				fbRecebe.bExecute := TRUE;
			END_IF
				
			fbRecebe(
				sSrvNetId:= '', 
				hSocket:= fbConection.hSocket, 
				cbLen:= SIZEOF(sRecebidoB), 
				pDest:= ADR(sRecebidoB), 
				bExecute:= , 
				tTimeout:= , 
				bBusy=> , 
				bError=> , 
				nErrId=> , 
				nRecBytes=> );
				
			IF fbRecebe.bError THEN
				fbConection(bEnable:= false);
			END_IF
				
			IF NOT fbRecebe.bBusy THEN
					
				IF fbRecebe.nRecBytes > 0 THEN
					//ajusta o que veio pra ficar como a gente quer
					sRecebido := LEFT(STR:= sRecebidoB, SIZE:=TO_INT(fbRecebe.nRecBytes));
					
					
					IF  '$02(103' = LEFT(STR:= sRecebido, SIZE:=5) THEN
						
						sTeste := sRecebido;
						sAjustado := DELETE(STR:= sRecebido, LEN:= 9, POS:= 0);
						sAjustado := LEFT(STR:= sAjustado, SIZE:= 5);
						rPeso := TO_REAL(sAjustado);
						
						xNovoResultado := TRUE;
						
						//ajusta no buffer
						FOR i := 9 TO 1 BY -1 DO
							stBuffer[i] := stBuffer[i-1];
						END_FOR
						
						stBuffer[0] := rPeso;
						
						iContador := iContador + 1;
					
					END_IF
				END_IF
				
				
				IF xResetContador THEN
					xResetContador := FALSE;
					iContador := 0;
				END_IF
				
				fbRecebe.bExecute := FALSE;
				fbRecebe();
				
			END_IF
			
		1://lenk
		
			xNovoResultado := FALSE;
			
			
			//conecta na tcp socket
			fbConection(
				sSrvNetID:= '', 
				nMode:= CONNECT_MODE_ENABLEDBG, 
				sRemoteHost:= ip, 
				nRemotePort:= 2306, 
				bEnable:= xConecta, 
				tReconnect:= T#1S, 
				bBusy=> , 
				bError=> , 
				nErrId=> , 
				hSocket=> , 
				eState=> );
				
				
			IF NOT fbConection.bBusy THEN
				xAuxOnline := xConecta;
				IF fbConection.bError THEN
					nErrId := fbConection.nErrId;
					xAuxOnline := FALSE;
				END_IF
			END_IF
			
			
			tofOffline(IN:= xAuxOnline, PT:= T#5S, Q=> xOnline, ET=> );
			
			
			//fica rodando o recebe pra ficar lendo caso aparece alguma coisa
			IF NOT fbRecebe.bExecute THEN
				fbRecebe.bExecute := TRUE;
			END_IF
				
			fbRecebe(
				sSrvNetId:= '', 
				hSocket:= fbConection.hSocket, 
				cbLen:= SIZEOF(sRecebidoB), 
				pDest:= ADR(sRecebidoB), 
				bExecute:= , 
				tTimeout:= , 
				bBusy=> , 
				bError=> , 
				nErrId=> , 
				nRecBytes=> );
				
			IF fbRecebe.bError THEN
				fbConection(bEnable:= false);
			END_IF
				
			IF NOT fbRecebe.bBusy THEN
					
				IF fbRecebe.nRecBytes > 0 THEN
					//ajusta o que veio pra ficar como a gente quer
					sRecebido := LEFT(STR:= sRecebidoB, SIZE:=TO_INT(fbRecebe.nRecBytes));
					
					
					sAjustado := REPLACE(STR1:= sRecebido, STR2:= '', L:= 2, P:=0 );
					rPeso := TO_REAL(LEFT(STR:= sAjustado, SIZE:=3));
					sAjustado := REPLACE(STR1:= sRecebido, STR2:= '', L:= 5, P:=0 );
					sAjustado := LEFT(STR:= sAjustado, SIZE:=3);
					
					raux := TO_REAL(sAjustado);
					IF raux <> 0 THEN
						rPeso := rPeso + raux/1000;
					END_IF
					
					xNovoResultado := TRUE;
					
					//ajusta no buffer
					FOR i := 9 TO 1 BY -1 DO
						stBuffer[i] := stBuffer[i-1];
					END_FOR
					
					stBuffer[0] := rPeso;
					
					iContador := iContador + 1;
					
				END_IF
				
					
			END_IF
				
			IF xResetContador THEN
				xResetContador := FALSE;
				iContador := 0;
			END_IF
				
				
			fbRecebe.bExecute := FALSE;
			fbRecebe();
				
			
	
	END_CASE

END_IF

END_FUNCTION_BLOCK

// POUs/Automatico/Aspercao/Balanca/FB_SalvaBalancaBanco
FUNCTION_BLOCK FB_SalvaBalancaBanco
VAR_INPUT
	stBalanca : st_Balanca;
	sNomeTabela : STRING;
	stHoraAhora : TIMESTRUCT;
END_VAR
VAR_OUTPUT
	xOcupado : BOOL;
END_VAR
VAR
	rPesoAnterior : REAL;
	rtMudouPeso : R_TRIG;
	xSalva : BOOL;
	
	fbPLCDB  : FB_PLCDBCmdEvt(sNetID := '', tTimeout := T#5S);
    sCmd          : STRING (1000); 
    aPara         : ST_ExpParameter;
	sAux 		  : STRING;
	saAux : ARRAY[0..50] OF STRING(80);//para gerar os comandos
	I	: INT;
END_VAR




rtMudouPeso(CLK:= rPesoAnterior <> stBalanca.rPeso, Q=> );
IF rtMudouPeso.q THEN
	rPesoAnterior := stBalanca.rPeso;
	xSalva := TRUE;
END_IF

//INSERT INTO `geral`.`quente` (`rPeso`, `timestamp`) VALUES ('1.1', '1');

IF xSalva THEN
	
	xOcupado := TRUE;
	
	FOR i:= 0 TO 50 DO
		saAux[i]:= '';
	END_FOR

	saAux[0] := ('INSERT INTO `geral`.`');
	saAux[1] := sNomeTabela;
	saAux[2] := ('` (`rPeso`, `timestamp`) VALUES ($'');
	saAux[3] := REAL_TO_STRING(stBalanca.rPeso);
	saAux[4] := ('$', $'');
	saAux[5] := (TO_STRING(stHoraAhora.wYear));
	saAux[6] := ('-');
	saAux[7] := (TO_STRING(stHoraAhora.wMonth));
	saAux[8] := ('-');
	saAux[9] := (TO_STRING(stHoraAhora.wDay));
	saAux[10] := (' ');
	saAux[11] := (TO_STRING(stHoraAhora.wHour));
	saAux[12] := (':');
	saAux[13] := (TO_STRING(stHoraAhora.wMinute));
	saAux[14] := (':');
	saAux[15] := (TO_STRING(stHoraAhora.wSecond));
	saAux[16] := ('$');');
	
	sCmd := F_ConcatArray1000(sArray:= saAux);
	
	aPara.eParaType := E_ExpParameterType.STRING_;
	aPara.nParaSize := SIZEOF(sAux);

	// call functionblock
	IF fbPLCDB.Execute(
		hDBID:= 1, 
		pExpression:= ADR(sCmd), 
		cbExpression:= SIZEOF(sCmd), 
		pData:= ADR(sAux), 
		cbData:= SIZEOF(sAux), 
		pParameter:= ADR(aPara), 
		cbParameter:= SIZEOF(aPara)) 
	THEN
		xSalva := FALSE;
		xOcupado := FALSE;
		IF NOT fbPLCDB.bError THEN
			//
		END_IF
	END_IF
END_IF

END_FUNCTION_BLOCK

// POUs/Automatico/Aspercao/Camaras/FB_Camaras
FUNCTION_BLOCK FB_Camaras
VAR_IN_OUT
	Camara : st_Camara;
	stControleValvulas : ARRAY[*] OF st_ControleValvula;
END_VAR
VAR_INPUT
	iCamara : INT;//numero da camara
	sNome	: STRING;//nome da camara
	sGuidAtual: STRING;// guid do processo que ela esta fazendo atualmente
	sValvulas : STRING;// valvula que estao nessa camara
	
	xCamaraTempOK	: BOOL; //Temperatura da camera esta OK
	xCamaraUmidOK	: BOOL; //Umidade da camera esta OK
	xAnelPressOK	: BOOL; //Pressao do anel esta OK
	xTanqueTempOK	: BOOL; //Temperatura do tanque esta OK
	
	stHoraAhora : TIMESTRUCT;
	xAmostra : BOOL; //amostra para o banco algumas variaveis ciclicamente
	
	xAtualizaValvulasCluster : BOOL;
END_VAR
VAR_OUTPUT
	sStatus : STRING;// status da camara
	iStatus : INT;//status da carama que vai para a ihm
	iQuantidadeDeCluster : INT;//Quantos cluster estao sendo usados
	iValvulaMestraMestra : INT;//a primeira valvula que liga na aspersao, so começa a contar o tempo depois que ela liga a primeira vez
END_VAR
VAR
	
	
	CamaraAnterior : st_Camara;
	i,k,l : INT;
	iValvulas 			: ARRAY[0..500] OF INT;
	rtSemGuid 			: R_TRIG;
	rtComecouAspercao 	: R_TRIG;
	rtTerminouAspercao 	: R_TRIG;
	xIniciouAspercao 	: BOOL;
	tonInicioAspercao 	: ton;
	xTerminouAspercao 	: BOOL;
	
	tonAmostra : TON;
	
    fbPLCDBCmd,fbPLCDBaspersao,fbPLCDBResfriamento,fbDBCmdAFCluster,fbDBInicioProcesso,fbDBFimProcesso,fbPLCDProtocolo : FB_PLCDBCmdEvt(sNetID := '', tTimeout := T#5S);
	
    sCmd          : STRING (1000); 
    aPara         : ST_ExpParameter;
	sAux 		  : STRING;
	
	xSalvaGrafico : BOOL;
	xSalvaEvento : BOOL;
	j : INT := 0;
	xSalvaResfriamento : BOOL;
	xSalvaFimResfriamento : BOOL;
	xSalvaInicioAspersao : BOOL;
	xSalvaFimAspersao : BOOL;
	
	rt_ComecouResfriamento : R_TRIG;
	
	xPegaInicioResfriamento : BOOL := TRUE;
	xPegaInicioAspersao : BOOL := TRUE;
	xPegaFimAspersao : BOOL;
	xAuxAspersao : BOOL;
	tonOnIniciaAAspersao : TON;
	
	fbSalvaEvento : ARRAY[0..15] OF FB_SalvaEventoRelatorio;
	rtCancelouValvula : R_TRIG;
		
	rtTemReferencia : R_TRIG;
	xFirstScan : BOOL := TRUE;
	
	xFinalizaValvulasDaCamara : BOOL;
		
	saAux : ARRAY[0..50] OF STRING(80);//para gerar os comandos
	
	iAux : INT;
	
	iNumeroDeClusters : INT := 30;
	
	xProtocolo1Etapa : BOOL;
	xComProcessoMasNaoIniciouValvula : BOOL;
	rtComGuid : R_TRIG;
	
	xTodasComecaram : BOOL;
	dtValvulaMestreMestre : DT;
	xIniciaSincronismo : BOOL;
	
	iOrdemCluster : ARRAY[0..100] OF INT;
	iEtapaAux,iValvulaMestreAux,iValvulaMestreMestreAux,iValvulaAux : INT;
	lrTonAux,lrToffAux : LREAL;
	rEtapasAux: ARRAY[1..10,1..3] OF LREAL;
	
	iDebug : INT;
	
	xPodeEntrar : BOOL;
	lrDiferencaTempo : LREAL;
	
	iClusterSalvando : INT;
	xSalvaONOFFCluster : BOOL;
	xStatusLigado : BOOL;
	
	tonSincornismo : TON_P;
	rtMomentoDeEntrada : R_TRIG;
	
	tTempoAteSinc : TIME;
	dtAux : DT;
	
	
	fbProcessoEmail : NT_StartProcess;
	sComando: STRING;
	xGeraRelatorio : BOOL;
	
	sGuidAnterior : STRING;
	
	xSalvaQueFoiArrancadoOProcesso : BOOL;
	xSalvaIniSemPeso : BOOL;
	xSalvaFimSemPeso : BOOL;
	
	iMaquinaIniciaSemPeso : INT;
	fbCriaGUID 	: FB_CreateGUID;
	guidCriado 	: Guid;
	
	xSalvaProtocolo : BOOL;
	
	rtValvulaMestreMestreSetada : R_TRIG;
	
	iClusterAux : INT;
	iAuxValvula : INT;
	tAux : TIME;
	
	tonPodeGerarRelatorio : TON;
	
	rtLigaTudo : r_trig;
	
	ton10s : TON;
	x10s : BOOL;
	ton2s : TON;
	x2s : BOOL;
	ton500ms : TON;
	x500ms : BOOL;
	
END_VAR

IF TRUE THEN	
	
	AjustaEntrada();

	SalvaGrafico();
	InicioPelaCamara();
	
	//so joga as referencias se a referencia for valida (pode ser so a primeira pq quando a primeira tiver toda tem)
	IF xFirstScan THEN
		FOR i := 0 TO 500 DO
			IF iValvulas[i] = 0 THEN
				EXIT;
			ELSE
				stControleValvulas[iValvulas[i]].EN.iValvulasAbertasCamara REF= Camara.config.iValvulasAbertasNaCamara;
				stControleValvulas[iValvulas[i]].EN.iMaxValvulasAbertasCamara := Camara.config.iMaxValvulasAbertasCamara;
			END_IF
		END_FOR
	END_IF
	
	//Ta com o nome do rt errado aqui, mas nao da pra criar um entao ne
	rtTemReferencia(CLK:= Camara.en.xFinalizaCamaraIHM, Q=> );
	
	IF (Camara.en.xApagaProcessoSupervisorio OR ((Camara.en.xFinalizaCamaraSupervisorio OR rtTemReferencia.q) AND xTerminouAspercao)) AND sGuidAtual <> '' THEN
		Camara.en.sGuidAtual := '';
		sGuidAtual := '';
		//Salva evetos
		xSalvaQueFoiArrancadoOProcesso := Camara.en.xApagaProcessoSupervisorio;
		xSalvaFimSemPeso := Camara.en.xFinalizaCamaraSupervisorio;
		xSalvaFimResfriamento := TRUE;
		//Tira os bits
		Camara.en.xApagaProcessoSupervisorio := FALSE;
		Camara.en.xFinalizaCamaraSupervisorio := FALSE;
		Camara.en.xFinalizaCamaraIHM := FALSE;
	END_IF
	
	
	//pra quando quer acabar a camara inteira mais rapido
	IF xFinalizaValvulasDaCamara THEN
		xIniciouAspercao := TRUE;
		xTerminouAspercao := TRUE;
		xFinalizaValvulasDaCamara := FALSE;
		FOR i := 0 TO 500 DO
			IF iValvulas[i] = 0 THEN
				EXIT;
			ELSE
				stControleValvulas[iValvulas[i]].en.xFinalizaInterno := TRUE;
			END_IF
		END_FOR
	END_IF
	
	
	rtComGuid(CLK:= sGuidAtual <> '', Q=> );
	IF rtComGuid.q THEN
		xComProcessoMasNaoIniciouValvula := TRUE;
		sGuidAnterior := sGuidAtual;
		Camara.sa.tHoraInicio := SYSTEMTIME_TO_DT(stHoraAhora);
	END_IF
	
	
	// da liga em todas as valvulas
	rtLigaTudo(CLK:= (Camara.en.xLigaTudoFisico AND NOT Camara.Config.xIgnoraBotaoFisico) OR Camara.en.xLigaTudoIHM OR Camara.en.xLigaTudoSupervisorio, Q=> );
	IF rtLigaTudo.Q THEN
		FOR i := 0 TO 500 DO
			IF iValvulas[i] = 0 THEN
				EXIT;
			ELSE
				stControleValvulas[iValvulas[i]].EN.stProtocolos[0].xSelecionado := TRUE;
			END_IF
		END_FOR
		
		IF Camara.Status.sOndeFoiIniciado = '' THEN
			IF Camara.en.xLigaTudoIHM THEN
				Camara.Status.sOndeFoiIniciado := 'IHM';
			END_IF
			IF Camara.en.xLigaTudoSupervisorio THEN
				Camara.Status.sOndeFoiIniciado := 'Supervisorio';
			END_IF
			IF (Camara.en.xLigaTudoFisico AND NOT Camara.Config.xIgnoraBotaoFisico) THEN
				Camara.Status.sOndeFoiIniciado := 'Botão fisico';
			END_IF
		END_IF
		
	END_IF
	
		
	//se a umidade e temp ta ok
	xCamaraTempOK := Camara.config.rMaxTempCamara >= Camara.en.rTempCamara AND Camara.en.rTempCamara >= Camara.config.rMinTempCamara;
	xCamaraUmidOK := Camara.config.rMaxUmidCamara >= Camara.en.rUmidadeCamara AND Camara.en.rUmidadeCamara >= Camara.config.rMinUmidCamara;
	
	
	//Ajusta valvulas, passa as informaçoes para o controle das valvulas e pega quando inciou a valvula
	FOR i := 0 TO 500 DO
		IF iValvulas[i] = 0 THEN
			EXIT;
		ELSE
			//passa o guid para as valvulas 
			stControleValvulas[iValvulas[i]].EN.GUID := sGuidAtual;
			//passa o ok para as valvulas
			stControleValvulas[iValvulas[i]].EN.xCamaraTempOK := xCamaraTempOK;
			stControleValvulas[iValvulas[i]].EN.xCamaraUmidOK := xCamaraUmidOK;
			stControleValvulas[iValvulas[i]].EN.xAnelPressOK := xAnelPressOK;
			stControleValvulas[iValvulas[i]].EN.xTanqueTempOK := xTanqueTempOK;	
			//passa o tempo maximo para a valvula nas camaras
			stControleValvulas[iValvulas[i]].EN.iTempoMaximoAspersao := Camara.config.iTempoMaximoAspersao;	
			//se o protocolo é por camara ai ele que passa pra valvula quem ela vai seguir
			IF Camara.config.xProtocoloPorCamara THEN
				// passa os protocolos para as valvulas, o liga ainda vai pela valvula aqui ele so seleciona os protocolos
				//o mesmo protocolo em todos pq a valvula nao pode escolher outro
				stControleValvulas[iValvulas[i]].EN.stProtocolos[0].DB := Camara.config.stProtocolos[Camara.config.iProtocoloEscolhido].DB;
				stControleValvulas[iValvulas[i]].EN.stProtocolos[1].DB := Camara.config.stProtocolos[Camara.config.iProtocoloEscolhido].DB;
				stControleValvulas[iValvulas[i]].EN.stProtocolos[2].DB := Camara.config.stProtocolos[Camara.config.iProtocoloEscolhido].DB;
				stControleValvulas[iValvulas[i]].EN.stProtocolos[3].DB := Camara.config.stProtocolos[Camara.config.iProtocoloEscolhido].DB;
				stControleValvulas[iValvulas[i]].EN.stProtocolos[4].DB := Camara.config.stProtocolos[Camara.config.iProtocoloEscolhido].DB;
			END_IF
			//pasa o tempo para parar a ventilação
			stControleValvulas[iValvulas[i]].EN.iSegDesligarVentilacao := Camara.config.iSegDesligarVentilacao;
			//pasa o nome da camara
			stControleValvulas[iValvulas[i]].EN.sNomeCamara := Camara.config.sNome;
			//Passa tempo antes de começar a aspergir
			stControleValvulas[iValvulas[i]].EN.rTempoEsperaAntesAspergir := Camara.Config.rTempoEsperaAntesAspergir;
		END_IF
	END_FOR
	
	
	
	
	
	DefineQuandoSalvaEvento();
	
	ContrlCluster();
	
	
	
	//Quando acabar o processo tem que resetar algumas coisas
	rtSemGuid(CLK:= sGuidAtual = '', Q=> );
	IF rtSemGuid.q THEN
		xGeraRelatorio := TRUE;
		FOR i := 0 TO 1000 DO
			Camara.en.rPesosFrio[i] := 0;
			Camara.en.rPesosQuente[i] := 0;
		END_FOR
	END_IF
	
	IF sGuidAtual = '' THEN
		xIniciouAspercao := FALSE;
		xTerminouAspercao := FALSE;
		xPegaInicioResfriamento := TRUE;
		Camara.sa.tHoraInicio :=  DT#1970-01-01-00:00;
		Camara.sa.tHoraTermina := DT#1970-01-01-00:00;
		Camara.Status.sOndeFoiIniciado := '';
	END_IF
	
	
	Status();
	AjustaSaida();
	controleLed();
	
	
	
	i := iDebug;
	
	
	xFirstScan := FALSE;
	
	

END_IF

ACTION AjustaSaidaPeV:

//PArte do principio que nao precisa desligar nenhum ventilador
FOR j := 1 TO 10 DO
	Camara.sa.xDesligaEvaporador[j] := FALSE;
END_FOR



FOR i := 0 TO iNumeroDeClusters DO
	FOR j := 0 TO 20 DO
		IF Camara.Clusters[i].En.iValvulas[j] = 0 THEN
			EXIT;
		ELSE
			//Pausas
			iAux := Camara.Clusters[i].En.iValvulas[j];
			stControleValvulas[iAux].EN.xPausaSincCluster := Camara.Clusters[i].Sa.xPausaValvula[j];
			stControleValvulas[iAux].EN.xPausaSincEntreCluster := Camara.Clusters[i].En.xPausaCluster;
			
			//Quando para a ventilação
			iValvulaMestreAux := Camara.Clusters[i].Sa.iValvulaMestre;
			//pasa para o cluster o sinal que tem que para a ventilação
			Camara.Clusters[i].Sa.xParaVentilacao := stControleValvulas[iValvulaMestreAux].SA.xParaVentilacao;
		END_IF
	END_FOR
	
	//Quando para cada evaporador
	FOR j := 1 TO 10 DO
		//Se o cluster quer parar e ta habilitado para parar esse evaporador ele joga true no desliga evaporador da camara
		IF Camara.Clusters[i].Sa.xParaVentilacao AND Camara.Clusters[i].En.xHabilitaEvaporador[j] THEN
			Camara.sa.xDesligaEvaporador[j] := TRUE;
		END_IF
		//Força o sinal em manual para testes
		IF Camara.Config.xManualDesligaEvaporador[j] THEN
			Camara.sa.xDesligaEvaporador[j] := Camara.Config.xSinalManualDesligaEvap[j];
		END_IF
	END_FOR
	
END_FOR
END_ACTION

ACTION AtualizaValvulasDosClusters:


FOR i := 0 TO 30 DO
	FOR j := 0 TO 20 DO
		Camara.Clusters[i].En.iValvulas[j] := 0;
	END_FOR
END_FOR



//aqui cada cluster recebe as valvulas que estao nele
FOR i := 0 TO 100 DO //quantidade de valvulas na camara
	IF iValvulas[i] = 0 THEN
		EXIT;
	ELSE
		FOR j := 0 TO 20 DO// quantidade de valvulas em 1 cluster
			iaux := stControleValvulas[iValvulas[i]].EN.iCluster;
			IF Camara.Clusters[iaux].En.iValvulas[j] = 0  THEN
				Camara.Clusters[iaux].En.iValvulas[j] := stControleValvulas[iValvulas[i]].EN.iIndexValvula;
				EXIT;
			END_IF
		END_FOR
	END_IF
END_FOR
END_ACTION

ACTION ContrlCamaras:



	
lrTonAux := Camara.Config.stProtocolos[Camara.Config.iProtocoloEscolhido].DB.ET01TON;
lrToffAux := Camara.Config.stProtocolos[Camara.Config.iProtocoloEscolhido].DB.ET01TOFF;

Camara.sa.lrTempototal := (lrTonAux*1000 + lrToffAux*1000*60);
IF Camara.config.iQuantidadeCamaras = 0 THEN
	Camara.config.iQuantidadeCamaras := 1;
END_IF
Camara.sa.lrTempoDeCadaBloco := (lrTonAux*1000 + lrToffAux*1000*60) / Camara.config.iQuantidadeCamaras;
Camara.sa.lrPosicaoDeEntrada := Camara.sa.lrTempoDeCadaBloco * Camara.config.iPosisaoCamara;

IF TIME_TO_LREAL(tonSincornismo.ET) < Camara.sa.lrPosicaoDeEntrada THEN
	tTempoAteSinc := LREAL_TO_TIME(Camara.sa.lrPosicaoDeEntrada) - tonSincornismo.ET;
ELSE
	tTempoAteSinc :=  (tonSincornismo.PT - tonSincornismo.ET) + LREAL_TO_TIME(Camara.sa.lrPosicaoDeEntrada);
END_IF

dtAux := TIME_TO_DT(tTempoAteSinc);

stControleValvulas[iValvulaMestraMestra].EN.tTempoAteSinc := tTempoAteSinc;

//Status de sincornizamento para a IHM/Supervisorio
IF iValvulaMestraMestra = 0 THEN
	Camara.status.sTempoAteCamaraEntrarNoSinc := 'Esperando 1ª Valvula';//se nao ligou a primeira ianda nao iniciou o role
ELSE
	IF stControleValvulas[iValvulaMestraMestra].EN.xPausaSincCamaras THEN
		Camara.status.sTempoAteCamaraEntrarNoSinc := REPLACE(STR1:= TO_STRING(dtAux), STR2:= '', L:= 15, P:=0);
	ELSE
		Camara.status.sTempoAteCamaraEntrarNoSinc := 'Sincronizada';
	END_IF
END_IF


//ton com autoreset, para de contar quando pausar pra nao perder o sincronismo, assim as camaras nao vao precisar resincronizar depois de voltar a pausa
tonSincornismo(IN:=TRUE, pt:=REAL_TO_TIME(Camara.sa.lrTempototal), PAUSE:= NOT xTanqueTempOK OR NOT xAnelPressOK);
IF tonSincornismo.q THEN
	//quando termina o ciclo ele da reset
	tonSincornismo(IN:=FALSE);
END_IF


IF iValvulaMestraMestra <> 0 THEN
	
	//Verifica se a valvula mestre mestre foi cancelada
	IF stControleValvulas[iValvulaMestraMestra].SA.iStatus = 9 THEN
		//Fica zerada pq tem que trocar 
		iValvulaMestraMestra := 0;
		
		//Se cancelou procura uma valvula em algum cluster que ja tenha iniciado para virar a mestra
		FOR i := 0 TO 500 DO
			// Se ela tiver aspergindo ou esperando pra aspergir é a mestra mestra facin
			IF stControleValvulas[iValvulas[i]].SA.iStatus = 5 OR stControleValvulas[iValvulas[i]].SA.iStatus = 6 THEN
				iValvulaMestraMestra := iValvulas[i];
				EXIT;
			END_IF 
		END_FOR
		
		//Se nao tem ninguem aberto em cima procura um que esteja em processo pelo menos
		IF iValvulaMestraMestra = 0 THEN
			FOR i := 0 TO 500 DO
				// Se ela tiver aspergindo ou esperando pra aspergir é a mestra mestra facin
				IF stControleValvulas[iValvulas[i]].SA.iStatus <> 9 AND stControleValvulas[iValvulas[i]].SA.iStatus <> 3
				AND stControleValvulas[iValvulas[i]].SA.iStatus <> 99 AND stControleValvulas[iValvulas[i]].SA.iStatus <> 4 THEN
					iValvulaMestraMestra := iValvulas[i];
					EXIT;
				END_IF 
			END_FOR
		END_IF
		
	
		
		//Se nos dois for de cima encontrou alguem ajusta, se nao nao tem ningume pra virar mestra mestra
		IF iValvulaMestraMestra <> 0 THEN
			stControleValvulas[iValvulaMestraMestra].EN.xPausaSincCamaras := NOT xIniciaSincronismo;
			
			iClusterAux := 0;
			//procura o cluster dessa valvula para tirar o pause dela
			FOR k := 1 TO iNumeroDeClusters DO
				//Se encontrou o cluster da valvula ele pula fora 
				IF iClusterAux <> 0 THEN
					EXIT;
				END_IF
				//se o cluster nao tem valvula pula ele e vai pro proximo
				IF Camara.Clusters[k].En.iValvulas[0] = 0 THEN
					//nao faz nada
				ELSE
					FOR l := 0 TO 20 DO
						//se ta em 0 nao usa e cabou as valvulas 
						IF Camara.Clusters[k].En.iValvulas[l] = 0 THEN
							EXIT;
						ELSE
							IF iValvulaMestraMestra = stControleValvulas[iValvulas[l]].EN.iIndexValvula THEN
								iClusterAux := k;
								EXIT;
							END_IF
						END_IF
					END_FOR
				END_IF
			END_FOR
			
					
			FOR l := 0 TO 20 DO
				//Procura a valvula mestra e tira a pausa dela se ela tiver
				IF Camara.Clusters[iClusterAux].En.iValvulas[l] = iValvulaMestraMestra THEN
					Camara.Clusters[iClusterAux].En.xPausaCluster := FALSE;
					Camara.Clusters[iClusterAux].sa.xPausaValvula[l] := FALSE;
					EXIT;
				END_IF
			END_FOR	
		ELSE
		//Se ainda ta sem mestra quer dizer que nao tem ninguem ligada ai zera os role
			//Se cancelou procura uma valvula em algum cluster que ja tenha iniciado para virar a mestra
			FOR i := 0 TO 500 DO
				IF iValvulas[i] = 0 THEN
					//Nao encontrou nenhuma pra pegar o lugar
					iValvulaMestraMestra := 0;
					xComProcessoMasNaoIniciouValvula := TRUE;
					
					FOR k := 1 TO iNumeroDeClusters DO
						//se o cluster nao tem valvula pula ele e vai pro proximo
						IF Camara.Clusters[k].En.iValvulas[0] = 0 THEN
							//nao faz nada
						ELSE
							Camara.Clusters[k].Sa.iValvulaMestre := 0;
							Camara.Clusters[k].Sa.iAbertas := 0;
							Camara.Clusters[k].En.iPosisaoCluster := 0;
							Camara.Clusters[k].i.iEtapaAnterior := 1;
							Camara.Clusters[k].En.xPausaCluster := FALSE;
							FOR l := 0 TO 20 DO
								Camara.Clusters[k].Sa.xLigadoAnterior[l] := 0;
								Camara.Clusters[k].Sa.xPausaValvula[l] := FALSE;
							END_FOR
						END_IF
					END_FOR
					
					//Zera a ordem dos cluster
					FOR i := 0 TO 100 DO
						iOrdemCluster[i] := 0;
					END_FOR
					
					//zera a hora de inicio de sincronia
					dtValvulaMestreMestre :=  DT#1970-01-01-00:00;
					xIniciaSincronismo := FALSE;
					EXIT;
				END_IF
			END_FOR
		END_IF
		
	END_IF




	
	//fica contando o tempo ate o momento que ele pode entrar, quando liberar ele ve se a valvula pode ligar, se ela pode ele tira o interlock
	//Camara.Clusters[i].i.TonMomentoDeEntrada(IN:=Camara.Clusters[i].i.xIniciaSincronismo,pt:=REAL_TO_TIME(Camara.Clusters[i].i.lrPosicaoDeEntrada));
	lrDiferencaTempo := TIME_TO_LREAL(tonSincornismo.ET) - Camara.sa.lrPosicaoDeEntrada;
	xPodeEntrar := lrDiferencaTempo > -100 AND lrDiferencaTempo < 100;
	rtMomentoDeEntrada(CLK:=xPodeEntrar AND iValvulaMestraMestra <> 0);
	IF rtMomentoDeEntrada.q AND stControleValvulas[iValvulaMestraMestra].EN.xPausaSincCamaras THEN
		//passa em todas as valvulas e diz que ta sem pausa de sin cam
		FOR i := 0 TO 500 DO
			IF iValvulas[i] = 0 THEN
				EXIT;
			ELSE
				// passa em todas as valvulas
				//joga todas em pausa por sincronismo quando da pausa por causa do sistema
				stControleValvulas[iValvulas[i]].EN.xPausaSincCamaras := FALSE;
			END_IF
		END_FOR
		
		//Encontra o cluster da master e tira a pausa entre cluster dela, mas coloca a pausa entre clusters nas outras
		iClusterAux := 0;
		FOR k := 1 TO iNumeroDeClusters DO
			Camara.Clusters[k].En.xPausaCluster := TRUE;
			IF Camara.Clusters[k].En.iValvulas[0] = 0 THEN
				//nao faz nada
			ELSE
				FOR l := 0 TO 20 DO
					//se ta em 0 nao usa e cabou as valvulas 
					IF Camara.Clusters[k].En.iValvulas[l] = 0 THEN
						EXIT;
					ELSE
						IF iValvulaMestraMestra = Camara.Clusters[k].En.iValvulas[l] THEN
							Camara.Clusters[k].En.xPausaCluster := FALSE;
						END_IF
					END_IF
				END_FOR
			END_IF
		END_FOR
		
		
	END_IF
	
	
	//se a mestre pausar significa que pausou a camara inteira, ai tem que parar todo mundo pra resincronizar com a camara quando voltar da pausa
	IF stControleValvulas[iValvulaMestraMestra].SA.xPausado THEN
		IF NOT xCamaraTempOK OR NOT xCamaraUmidOK THEN
			FOR i := 0 TO 500 DO
				IF iValvulas[i] = 0 THEN
					EXIT;
				ELSE
					// passa em todas as valvulas
					//joga todas em pausa por sincronismo quando da pausa por causa do sistema
					//So tem que resincrozinar se for alguma coisa especifica da camara, que se nao parou todo mundo e ja eras né
					stControleValvulas[iValvulas[i]].EN.xPausaSincCamaras := TRUE;
				END_IF
			END_FOR
		END_IF
	END_IF
	
	
END_IF
END_ACTION

ACTION ContrlCluster:



IF xAtualizaValvulasCluster OR Camara.en.xAtualizaValvulasCluster THEN
	AtualizaValvulasDosClusters();
	xAtualizaValvulasCluster := FALSE;
	Camara.en.xAtualizaValvulasCluster := FALSE;
END_IF

IF sGuidAtual = '' THEN
	Camara.sa.xPodeIniciar := FALSE;
	FOR i := 0 TO 100 DO
		iOrdemCluster[i] := 0;
	END_FOR
END_IF


ContrlCamaras();
ContrlEntreClusters();


//roda todos os clusters
FOR i := 1 TO iNumeroDeClusters DO
	//se o cluster nao tem valvula pula ele e vai pro proximo
	IF Camara.Clusters[i].En.iValvulas[0] = 0 THEN
		//nao faz nada
	ELSE
		//aqui ele passa em cada um dos clusters
		
		Camara.Clusters[i].En.rTempoEntreValvulas := 0.25;
		
		//se a camara ta liberada pra iniciar libera as valvula mestra
		IF Camara.sa.xPodeIniciar THEN
			iValvulaMestreAux := Camara.Clusters[i].Sa.iValvulaMestre;
			stControleValvulas[iValvulaMestreAux].EN.xPausaSincCamaras := FALSE;
		END_IF
		
		//se nao tem guid deixa tudo resetado 
		IF sGuidAtual = '' THEN
			Camara.Clusters[i].Sa.iValvulaMestre := 0;
			Camara.Clusters[i].Sa.iAbertas := 0;
			Camara.Clusters[i].En.iPosisaoCluster := 0;
			Camara.Clusters[i].i.iEtapaAnterior := 1;
			Camara.Clusters[i].En.xPausaCluster := FALSE;
			iValvulaMestraMestra := 0;
			
			FOR j := 0 TO 20 DO
				Camara.Clusters[i].Sa.xLigadoAnterior[j] := 0;
				Camara.Clusters[i].Sa.xPausaValvula[j] := FALSE;
			END_FOR
			
			//zera a hora de inicio de sincronia
			dtValvulaMestreMestre :=  DT#1970-01-01-00:00;
			xIniciaSincronismo := FALSE;
		ELSE
			
		
			//Verifica se a valvula mestre do cluster nao foi cancelada
			IF stControleValvulas[Camara.Clusters[i].Sa.iValvulaMestre].SA.iStatus = 9 THEN
				
				Camara.Clusters[i].Sa.iValvulaMestre := 0;
				//Se cancelou procura uma valvula no cluster que ja tenha iniciado para virar a mestra
				FOR j := 0 TO 20 DO
					IF stControleValvulas[Camara.Clusters[i].En.iValvulas[j]].SA.iStatus = 5 OR stControleValvulas[Camara.Clusters[i].En.iValvulas[j]].SA.iStatus = 6 THEN
						
						Camara.Clusters[i].Sa.iValvulaMestre := Camara.Clusters[i].En.iValvulas[j];
						stControleValvulas[Camara.Clusters[i].Sa.iValvulaMestre].EN.xPausaSincCamaras := NOT xIniciaSincronismo;
						Camara.Clusters[i].sa.xPausaValvula[j] := FALSE;
						EXIT;
					END_IF 
				END_FOR
				
				//Se nao encontrou procura uma que esteja pausada msm
				IF Camara.Clusters[i].Sa.iValvulaMestre = 0 THEN
					FOR j := 0 TO 20 DO
						iAux := Camara.Clusters[i].En.iValvulas[j];
						
						IF stControleValvulas[iaux].SA.iStatus <> 9 AND stControleValvulas[iaux].SA.iStatus <> 3
						AND stControleValvulas[iaux].SA.iStatus <> 99 AND stControleValvulas[iaux].SA.iStatus <> 4 THEN
						
							Camara.Clusters[i].Sa.iValvulaMestre := iaux;
							stControleValvulas[iaux].EN.xPausaSincCamaras := NOT xIniciaSincronismo;
							//Ja que nao tem ninguem rodando pausa todo o cluster ate sincronizar
							Camara.Clusters[i].En.xPausaCluster := TRUE;
							Camara.Clusters[i].sa.xPausaValvula[j] := FALSE;
							EXIT;
						END_IF 
					END_FOR 
				END_IF
				
				
				//se ta 0 é pq nao tem ninguem pra ficar no lugar dela ai pula fora
				IF Camara.Clusters[i].Sa.iValvulaMestre = 0 THEN
					//Nao tem nenhuma outra pra virar a mestra desse cluster
					Camara.Clusters[i].Sa.iValvulaMestre := 0;
					//Ve qual a posição desse cluster e libera ela pra alguem usar
					FOR k := 0 TO 100 DO
						IF iOrdemCluster[k] = i THEN
							iOrdemCluster[k] := 0;
							EXIT;
						END_IF
					END_FOR
				END_IF
			END_IF
			
			
			
			
		
		
			
			Camara.Clusters[i].Sa.xAlgumaValvulaAberta := FALSE;
			//ve se alguma valvula foi pra em processo e define a valvula mestre se for o caso
			FOR j := 0 TO 20 DO
				//se ta em 0 nao usa e cabou as valvulas 
				IF Camara.Clusters[i].En.iValvulas[j] = 0 THEN
					EXIT;
				ELSE
					
					iaux := Camara.Clusters[i].En.iValvulas[j];
					//Se a valvula foi cancelada reinicia as config dela
					IF stControleValvulas[iAux].SA.iStatus = 9 THEN
						Camara.Clusters[i].sa.xPausaValvula[j] := FALSE;
						Camara.Clusters[i].sa.xLigadoAnterior[j] := FALSE;
					END_IF
					
					//Se for a valvula mestra nao pode ter a pausa do cluster//08/02/2024
					IF iAux = Camara.Clusters[i].Sa.iValvulaMestre THEN
						Camara.Clusters[i].Sa.xPausaValvula[j] := FALSE;
					END_IF
				
				
					//ve se a valvula mestra ja abriu, quando ela abrir pode liberar a sincronia
					IF stControleValvulas[iValvulaMestraMestra].SA.xValvulaAberta AND iValvulaMestraMestra <> 0 THEN
						xIniciaSincronismo := TRUE;
					END_IF
					//passa a hora de inicio de sincronia 
					Camara.Clusters[i].i.dthrInicioValMestre := dtValvulaMestreMestre;
					Camara.Clusters[i].i.xIniciaSincronismo := xIniciaSincronismo;
										
					
				
					//Ve se tem alguma valvula aberta para salvar no ton toff
					Camara.Clusters[i].Sa.xAlgumaValvulaAberta := Camara.Clusters[i].Sa.xAlgumaValvulaAberta OR stControleValvulas[iAux].SA.xValvulaAberta;
					//se entrou em processo e nao ta cancelada define o que vai rolar com ele
					IF stControleValvulas[iAux].SA.iStatus <> 9 AND stControleValvulas[iAux].SA.xEmProcesso <> Camara.Clusters[i].sa.xLigadoAnterior[j] THEN
						Camara.Clusters[i].sa.xLigadoAnterior[j] := stControleValvulas[iAux].SA.xEmProcesso;
						//se essa valvula ligou e nao foi definido o mestre ela é o mestre
						IF Camara.Clusters[i].Sa.iValvulaMestre = 0 THEN
							Camara.Clusters[i].Sa.iValvulaMestre := iaux;
							//manda tru aqui que ali em baixo nao pode pausar a mestre
							Camara.Clusters[i].i.xHEaMestre := TRUE;
							//Se é a mestre que liga entao tem que pausar o cluster pra sincronizar
							Camara.Clusters[i].En.xPausaCluster := TRUE;
							
							//pausa ela ate a camara dizer que pode entrar, mas so se nao tiver começado o sincronismo
							stControleValvulas[iAux].EN.xPausaSincCamaras := NOT xIniciaSincronismo;
							
							// se true o de baixo, ele é a primeira valvula a ligar no role, a valvula mestre mestre
							IF xComProcessoMasNaoIniciouValvula THEN
								//A mestra mestra nao para pra sincronizar entre clusters
								Camara.Clusters[i].En.xPausaCluster := FALSE;
								//aqui ele vai ver se o protocolo tem mais de 1 etapa assim ele decide como vai funcionar
								xComProcessoMasNaoIniciouValvula := FALSE;
								//se o total de ciclos for maior que o numero de ciclos da 1 etapa ele tem mais de 1 etapa
								xProtocolo1Etapa := NOT (stControleValvulas[iAux].SA.iTotalDeCiclos > stControleValvulas[iAux].EN.stProtoEscolhido.DB.ET01NC);
								//ve a hora que ligou a primeira valvula e usa isso pra controlar o cluster das outras	
								dtValvulaMestreMestre := SYSTEMTIME_TO_DT(Camara.en.stHoraAgora);
								//salva quem é a valvula mestra mestra para quando ela ligar iniciar o sincronismo da galera
								iValvulaMestraMestra := iaux;
							END_IF
							
							//Ve qual a posição desse cluster
							FOR k := 0 TO 100 DO
								IF iOrdemCluster[k] = 0 THEN
									iOrdemCluster[k] := i;
									EXIT;
								END_IF
							END_FOR
							//salva a posição no cluster tb
							Camara.Clusters[i].En.iPosisaoCluster := k;
							
						END_IF
						
						//aqui so acontece quando muda o estado da valvula
						IF xProtocolo1Etapa THEN
							IF Camara.Clusters[i].i.xHEaMestre THEN
								Camara.Clusters[i].i.xHEaMestre := FALSE;
								Camara.Clusters[i].sa.xPausaValvula[j] := FALSE;
							ELSE
								//ela nao sendo o mestre tem que esperar pra ligar junto com ele
								Camara.Clusters[i].sa.xPausaValvula[j] := TRUE;
							END_IF
						ELSE
							//se ele tem mais de 1 etapa tem que fazer todos esperarem ate todos estarem na mesma etapa
							Camara.Clusters[i].sa.xPausaValvula[j] := TRUE;
							//ve se todas ja começaram, se ja começaram tira o pause de todas e pode partir
							xTodasComecaram := TRUE;
							FOR k := 0 TO 20 DO
								IF Camara.Clusters[i].En.iValvulas[k] = 0 THEN
									EXIT;
								END_IF
								xTodasComecaram := xTodasComecaram AND Camara.Clusters[i].sa.xLigadoAnterior[k];
							END_FOR
						END_IF
						
					END_IF
					
					Camara.Clusters[i].i.btONOFFCluster(CLK:=Camara.Clusters[i].Sa.xAlgumaValvulaAberta, Q=> );
					IF Camara.Clusters[i].i.btONOFFCluster.q THEN
						xSalvaONOFFCluster := TRUE;
						iClusterSalvando := i;
						xStatusLigado := Camara.Clusters[i].Sa.xAlgumaValvulaAberta;
					END_IF
					
					SalvaAbreEFechaNoCluster();
					
					
				END_IF
				
				//aqui so aplica se o protocolo for com mais de 1 etapa
				IF xTodasComecaram THEN
					//o todas começaram so serve para quando o cluster tem mais de 1 etapa
					xTodasComecaram := FALSE;
					FOR j := 0 TO 20 DO
						IF Camara.Clusters[i].En.iValvulas[j] = 0 THEN
							EXIT;
						ELSE
							Camara.Clusters[i].sa.xPausaValvula[j] := FALSE;
						END_IF
					END_FOR
				END_IF
				
				
				// quando a master liga ele tira o pause das outras
				// e faz no trigger pq se o cara ligar uma valvula quando a master ta na metade do liga ela vai ficar atrasada em relação as outras
				Camara.Clusters[i].i.rtMasterAbriu(CLK:= stControleValvulas[Camara.Clusters[i].Sa.iValvulaMestre].SA.xValvulaAberta);
				IF Camara.Clusters[i].i.rtMasterAbriu.q AND xProtocolo1Etapa THEN
					Camara.Clusters[i].i.xAjustaCascata := TRUE;
					iAux := 0;
					//conta quantas valvulas ja abriram
					FOR j := 0 TO 20 DO
						ivalvulaAux := Camara.Clusters[i].En.iValvulas[j];
						IF ivalvulaAux = 0 THEN
							EXIT;
						ELSE
							IF stControleValvulas[iValvulaAux].SA.xEmProcesso AND NOT Camara.Clusters[i].Sa.xPausaValvula[j] THEN
								iAux := iAux + 1;
							END_IF
						END_IF
					END_FOR
					Camara.Clusters[i].i.tTempoEsperaAntesCascata := REAL_TO_TIME(Camara.Clusters[i].En.rTempoEntreValvulas*1000*(iAux-1));
				END_IF
				
				//conta o tempo para ajustar a cascata de liga
				Camara.Clusters[i].i.tonAjusteTempoCascata(IN := Camara.Clusters[i].i.xAjustaCascata,PT := Camara.Clusters[i].i.tTempoEsperaAntesCascata);
				IF Camara.Clusters[i].i.tonAjusteTempoCascata.q THEN
					Camara.Clusters[i].i.xAjustaCascata := FALSE;
					Camara.Clusters[i].i.xRodaCascata := TRUE;
				END_IF
				
				//se pode rodar a cascata ele conta o tempo dele e vai para a proxima valvula para abrir ela
				Camara.Clusters[i].i.tonCascata(IN := Camara.Clusters[i].i.xRodaCascata,PT := REAL_TO_TIME(Camara.Clusters[i].En.rTempoEntreValvulas*1000));
				IF Camara.Clusters[i].i.tonCascata.Q THEN
					//ton com autoreset
					Camara.Clusters[i].i.tonCascata(IN := FALSE);
					
					FOR j := 0 TO 20 DO
						IF Camara.Clusters[i].En.iValvulas[j] = 0 THEN
							//se nao encontrou a proxima valvula para mandar abrir cabou
							Camara.Clusters[i].i.xRodaCascata := FALSE;
							EXIT;
						ELSE
							//encontra uma valvula pausada esperando para começar, e libera ela
							IF Camara.Clusters[i].sa.xPausaValvula[j] THEN
								Camara.Clusters[i].sa.xPausaValvula[j] := FALSE;
								EXIT;
							END_IF
						END_IF
					END_FOR
				END_IF
				
				
			END_FOR
		END_IF
	END_IF
END_FOR
















AjustaSaidaPeV();
END_ACTION

ACTION ContrlEntreClusters:
//calcula quantos cluster estao sendo usados
//roda todos os clusters
iQuantidadeDeCluster := 0;
FOR i := 0 TO iNumeroDeClusters DO
	//se o cluster nao tem valvula pula ele e vai pro proximo
	IF Camara.Clusters[i].En.iValvulas[0] = 0 THEN
		//nao faz nada
	ELSE
		iQuantidadeDeCluster := iQuantidadeDeCluster + 1;
	END_IF
END_FOR
iQuantidadeDeCluster := iQuantidadeDeCluster + Camara.config.iOffSetCluster;


//roda todos os clusters
FOR i := 0 TO iNumeroDeClusters DO
	//se o cluster nao tem valvula pula ele e vai pro proximo
	IF Camara.Clusters[i].En.iValvulas[0] = 0 THEN
		//nao faz nada
	ELSE
	//aqui passa em todos os cluster
		//variais variaveis aux pq o twincat nao funciona direito e nao lançam a 4026
		//usa a valvula mestre mestre para definir os tempo e quando cada um entra, mas para saber se mudou de etapa tem que usar a valvula mestre do cluster
		

		iValvulaMestreMestreAux := iValvulaMestraMestra;
		iValvulaMestreAux := Camara.Clusters[i].Sa.iValvulaMestre;
		IF stControleValvulas[iValvulaMestreAux].SA.iEtapaAtual = 0 THEN
			iEtapaAux := 1;
		ELSE
			iEtapaAux := stControleValvulas[iValvulaMestreAux].SA.iEtapaAtual;
		END_IF
		rEtapasAux := stControleValvulas[iValvulaMestreMestreAux].SA.rEtapasSemMudar;
		lrTonAux := rEtapasAux[iEtapaAux,1];
		lrToffAux := rEtapasAux[iEtapaAux,2];
		Camara.Clusters[i].i.lrTempototal := (lrTonAux*1000 + lrToffAux*1000*60);
		
		IF iQuantidadeDeCluster <> 0 THEN
			Camara.Clusters[i].i.lrTempoDeCadaBloco := (lrTonAux*1000 + lrToffAux*1000*60) / iQuantidadeDeCluster;
		END_IF
		
		Camara.Clusters[i].i.lrPosicaoDeEntrada := Camara.Clusters[i].i.lrTempoDeCadaBloco * Camara.Clusters[i].En.iPosisaoCluster;
		
		//ton com autoreset, para de contar quando pausar pra nao perder o sincronismo
		Camara.Clusters[i].i.tonSincornismo(IN:=Camara.Clusters[i].i.xIniciaSincronismo,pt:=REAL_TO_TIME(Camara.Clusters[i].i.lrTempototal),
											PAUSE:= stControleValvulas[iValvulaMestreMestreAux].SA.xPausadoSemSin);
		IF Camara.Clusters[i].i.tonSincornismo.q THEN
			//quando termina o ciclo ele da reset nos 2 
			Camara.Clusters[i].i.tonSincornismo(IN:=FALSE);
			Camara.Clusters[i].i.TonMomentoDeEntrada(IN:=FALSE);
		END_IF
		
		
		//quando inicia parte do principio que nenhum cluster esta sincronizado, entao bota todo mundo parado
		Camara.Clusters[i].i.rtIniciaSincronismo(CLK:=Camara.Clusters[i].i.xIniciaSincronismo);
		Camara.Clusters[i].i.rtTrocouEtapa(CLK:=iEtapaAux <> Camara.Clusters[i].i.iEtapaAnterior);
		IF Camara.Clusters[i].i.rtIniciaSincronismo.q OR Camara.Clusters[i].i.rtTrocouEtapa.q THEN
			Camara.Clusters[i].En.xPausaCluster := TRUE;
			//atualiza etapa
			Camara.Clusters[i].i.iEtapaAnterior := iEtapaAux;
		END_IF
		
		
		//fica contando o tempo ate o momento que ele pode entrar, quando liberar ele ve se a valvula pode ligar, se ela pode ele tira o interlock
		//Camara.Clusters[i].i.TonMomentoDeEntrada(IN:=Camara.Clusters[i].i.xIniciaSincronismo,pt:=REAL_TO_TIME(Camara.Clusters[i].i.lrPosicaoDeEntrada));
		lrDiferencaTempo := TIME_TO_LREAL(Camara.Clusters[i].i.tonSincornismo.ET) - Camara.Clusters[i].i.lrPosicaoDeEntrada;
		xPodeEntrar := lrDiferencaTempo > -100 AND lrDiferencaTempo < 100 AND Camara.Clusters[i].i.xIniciaSincronismo;
		Camara.Clusters[i].i.rtMomentoDeEntrada(CLK:=xPodeEntrar AND stControleValvulas[iValvulaMestreAux].SA.xNaoLigoSoPorSincETC);
		IF Camara.Clusters[i].i.rtMomentoDeEntrada.q THEN
			Camara.Clusters[i].En.xPausaCluster := FALSE;
		END_IF
		
		
		
		IF TIME_TO_LREAL(Camara.Clusters[i].i.tonSincornismo.ET) < Camara.Clusters[i].i.lrPosicaoDeEntrada THEN
			tAux := LREAL_TO_TIME(Camara.Clusters[i].i.lrPosicaoDeEntrada) - Camara.Clusters[i].i.tonSincornismo.ET;
		ELSE
			tAux :=  (Camara.Clusters[i].i.tonSincornismo.PT - Camara.Clusters[i].i.tonSincornismo.ET) + LREAL_TO_TIME(Camara.Clusters[i].i.lrPosicaoDeEntrada);
		END_IF
		
		//Passa quanto tempo falta para sincronizar
		FOR j := 0 TO 20 DO
			iAuxValvula := Camara.Clusters[i].En.iValvulas[j];
			IF iAuxValvula = 0 THEN
				EXIT;
			ELSE	
				//A mestra mestra tem outro role, e so pode passar o tempo pras valvulas depois da mestra mestra ter iniciado
				IF iAuxValvula <> Camara.sa.iValvulaMestraMestra AND NOT stControleValvulas[iValvulaMestreMestreAux].SA.xPausadoSemSin THEN
					IF Camara.Clusters[i].En.xPausaCluster THEN
						stControleValvulas[iAuxValvula].EN.tTempoAteSinc := tAux;
					ELSE
						//Um valor bem alto que não é pra considerar
						stControleValvulas[iAuxValvula].EN.tTempoAteSinc := T#10H;
					END_IF
				END_IF
			END_IF
		END_FOR
		
	END_IF
END_FOR












i := iDebug;
END_ACTION

ACTION SalvaAbreEFechaNoCluster:





IF xSalvaONOFFCluster AND iClusterSalvando = i AND FALSE THEN
	
	FOR k:= 0 TO 50 DO
		saAux[k]:= '';
	END_FOR
	
	//INSERT INTO `geral`.`clusteronoff` (`Cluster`, `Camara`, `Processo`, `Ligado`, `timestamp`) VALUES ('1', '1', '1', '1', '1');

	
	saAux[0] := ('INSERT INTO `geral`.`clusteronoff` (`Cluster`, `Camara`,');
	saAux[1] := (' `Processo`, `Ligado`, `timestamp`) VALUES ($'');
	saAux[2] := TO_STRING(iClusterSalvando);
	saAux[3] := ('$', $'');
	saAux[4] := (sNome);
	saAux[5] := ('$', $'');
	saAux[8] := (sGuidAtual);
	saAux[9] := ('$', $'');
	IF xStatusLigado THEN
		saAux[10] := '1';
	ELSE
		saAux[10] := '0';
	END_IF
	saAux[11] := ('$', $'');
	
	saAux[12] := (TO_STRING(camara.en.stHoraAgora.wYear));
	saAux[13] := ('-');
	saAux[14] := (TO_STRING(camara.en.stHoraAgora.wMonth));
	saAux[15] := ('-');
	saAux[16] := (TO_STRING(camara.en.stHoraAgora.wDay));
	saAux[17] := (' ');
	saAux[18] := (TO_STRING(camara.en.stHoraAgora.wHour));
	saAux[19] := (':');
	saAux[20] := (TO_STRING(camara.en.stHoraAgora.wMinute));
	saAux[21] := (':');
	saAux[22] := (TO_STRING(camara.en.stHoraAgora.wSecond));
	saAux[23] := ('$');');
	
	sCmd := F_ConcatArray1000(sArray:= saAux);
	
	aPara.eParaType := E_ExpParameterType.STRING_;
	aPara.nParaSize := SIZEOF(sAux);

	// call functionblock
	IF fbDBCmdAFCluster.Execute(
		hDBID:= 1, 
		pExpression:= ADR(sCmd), 
		cbExpression:= SIZEOF(sCmd), 
		pData:= ADR(sAux), 
		cbData:= SIZEOF(sAux), 
		pParameter:= ADR(aPara), 
		cbParameter:= SIZEOF(aPara)) 
	THEN
		xSalvaONOFFCluster := FALSE;
		iClusterSalvando := 0;
	END_IF
END_IF
END_ACTION

ACTION DefineQuandoSalvaEvento:


//Anel OK
fbSalvaEvento[1].xInicio := sGuidAtual <> '' AND xIniciouAspercao AND NOT xTerminouAspercao AND NOT xAnelPressOK;
//Temp Tanque OK
fbSalvaEvento[2].xInicio := sGuidAtual <> '' AND xIniciouAspercao AND NOT xTerminouAspercao AND NOT xTanqueTempOK;
//Temp Camara OK
fbSalvaEvento[3].xInicio := sGuidAtual <> '' AND xIniciouAspercao AND NOT xTerminouAspercao AND NOT xCamaraTempOK;
//Camara Umid OK
fbSalvaEvento[4].xInicio := sGuidAtual <> '' AND xIniciouAspercao AND NOT xTerminouAspercao AND NOT xCamaraUmidOK;



//Pega quando cancelou ou quando iniciou o resfriamento
FOR i := 0 TO 500 DO
	IF iValvulas[i] = 0 THEN
		EXIT;
	ELSE		
		IF xPegaInicioResfriamento AND (stControleValvulas[iValvulas[i]].SA.iStatus = 5 OR stControleValvulas[iValvulas[i]].SA.iStatus = 6) THEN
			xSalvaResfriamento := TRUE;
			xPegaInicioResfriamento := FALSE;
		END_IF
	END_IF
END_FOR




//Ve se terminou, so vai consderar se todos tiverem terminado
//esse sinal ´eo que libera para o camara ser tirada 
IF xIniciouAspercao AND NOT xTerminouAspercao THEN
	xTerminouAspercao := TRUE;
	FOR i := 0 TO 500 DO
		IF iValvulas[i] = 0 THEN
			EXIT;
		ELSE
			IF NOT (stControleValvulas[iValvulas[i]].SA.iStatus = 3 OR stControleValvulas[iValvulas[i]].SA.iStatus = 9) THEN //Finalizado ou cancelado
				xTerminouAspercao := FALSE;
			END_IF
		END_IF
	END_FOR	
END_IF


FOR i := 0 TO 30 DO
	camara.sa.iValvulas[i] := iValvulas[i];
END_FOR


//Ve se ja iniciou a asperção
IF NOT xIniciouAspercao THEN
	FOR i := 0 TO 500 DO
		IF iValvulas[i] = 0 THEN
			EXIT;
		ELSE// se tiver no processo de aspersao ou cancelado ele considera que ta aspergindo
			IF (stControleValvulas[iValvulas[i]].SA.iStatus = 5 OR stControleValvulas[iValvulas[i]].SA.iStatus = 6 OR stControleValvulas[iValvulas[i]].SA.iStatus = 9) THEN //Executando
				xIniciouAspercao := TRUE;
			END_IF
		END_IF
	END_FOR	
END_IF
InicioAspercao();


rtComecouAspercao(CLK:= xIniciouAspercao, Q=> );
IF rtComecouAspercao.q THEN
	xSalvaInicioAspersao := TRUE;
END_IF
InicioResfriamento();


rtTerminouAspercao(CLK:= xTerminouAspercao, Q=> );
IF rtTerminouAspercao.q THEN
	xSalvaFimAspersao := TRUE;
END_IF
fimAspersao();


IF xSalvaQueFoiArrancadoOProcesso THEN
	xSalvaQueFoiArrancadoOProcesso := FALSE;
	fbSalvaEvento[8].xInicio := TRUE;
	EventosRelatorio();
	fbSalvaEvento[8].xInicio := FALSE;
END_IF

IF xSalvaIniSemPeso THEN
	xSalvaIniSemPeso := FALSE;
	fbSalvaEvento[9].xInicio := TRUE;
	EventosRelatorio();
	fbSalvaEvento[9].xInicio := FALSE;
END_IF

IF xSalvaFimSemPeso THEN
	xSalvaFimSemPeso := FALSE;
	fbSalvaEvento[10].xInicio := TRUE;
	EventosRelatorio();
	fbSalvaEvento[10].xInicio := FALSE;
END_IF


//Salva o nome do protocolo no processo
rtValvulaMestreMestreSetada(CLK:= iValvulaMestraMestra <> 0, Q=> );
IF rtValvulaMestreMestreSetada.q THEN
	xSalvaProtocolo := TRUE;
END_IF
SalvaProtocolo();


FimResfriamento();
EventosRelatorio();
GeraRelatorio();


//Aqui o bloco que salva quando o protocolo foi cancelado recebe um fim para salvar no banco certinho
fbSalvaEvento[5].xInicio := FALSE;
END_ACTION

ACTION EventosRelatorio:
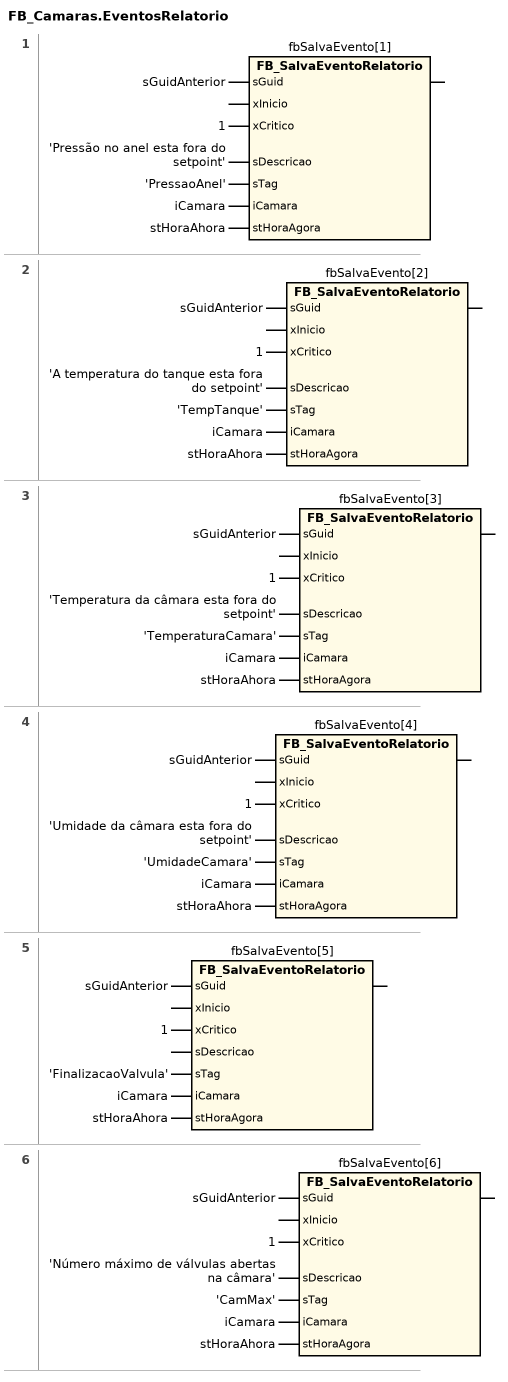
// NETWORK 1
fbSalvaEvento[1](
    sGuid := sGuidAnterior,
    xCritico := 1,
    sDescricao := 'Pressão no anel esta fora do setpoint',
    sTag := 'PressaoAnel',
    iCamara := iCamara,
    stHoraAgora := stHoraAhora); // FB_SalvaEventoRelatorio

// NETWORK 2
fbSalvaEvento[2](
    sGuid := sGuidAnterior,
    xCritico := 1,
    sDescricao := 'A temperatura do tanque esta fora do setpoint',
    sTag := 'TempTanque',
    iCamara := iCamara,
    stHoraAgora := stHoraAhora); // FB_SalvaEventoRelatorio

// NETWORK 3
fbSalvaEvento[3](
    sGuid := sGuidAnterior,
    xCritico := 1,
    sDescricao := 'Temperatura da câmara esta fora do setpoint',
    sTag := 'TemperaturaCamara',
    iCamara := iCamara,
    stHoraAgora := stHoraAhora); // FB_SalvaEventoRelatorio

// NETWORK 4
fbSalvaEvento[4](
    sGuid := sGuidAnterior,
    xCritico := 1,
    sDescricao := 'Umidade da câmara esta fora do setpoint',
    sTag := 'UmidadeCamara',
    iCamara := iCamara,
    stHoraAgora := stHoraAhora); // FB_SalvaEventoRelatorio

// NETWORK 5
fbSalvaEvento[5](
    sGuid := sGuidAnterior,
    xCritico := 1,
    sTag := 'FinalizacaoValvula',
    iCamara := iCamara,
    stHoraAgora := stHoraAhora); // FB_SalvaEventoRelatorio

// NETWORK 6
fbSalvaEvento[6](
    sGuid := sGuidAnterior,
    xCritico := 1,
    sDescricao := 'Número máximo de válvulas abertas na câmara',
    sTag := 'CamMax',
    iCamara := iCamara,
    stHoraAgora := stHoraAhora); // FB_SalvaEventoRelatorio

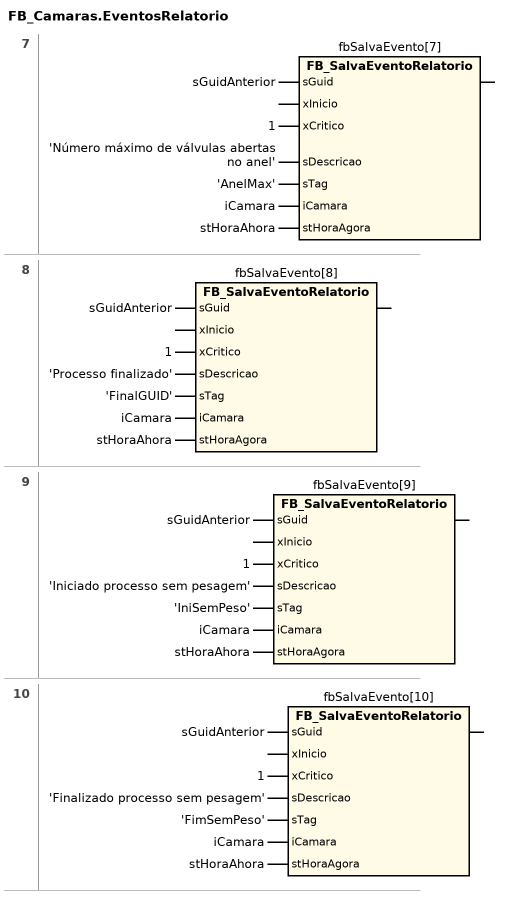
// NETWORK 7
fbSalvaEvento[7](
    sGuid := sGuidAnterior,
    xCritico := 1,
    sDescricao := 'Número máximo de válvulas abertas no anel',
    sTag := 'AnelMax',
    iCamara := iCamara,
    stHoraAgora := stHoraAhora); // FB_SalvaEventoRelatorio

// NETWORK 8
fbSalvaEvento[8](
    sGuid := sGuidAnterior,
    xCritico := 1,
    sDescricao := 'Processo finalizado',
    sTag := 'FinalGUID',
    iCamara := iCamara,
    stHoraAgora := stHoraAhora); // FB_SalvaEventoRelatorio

// NETWORK 9
fbSalvaEvento[9](
    sGuid := sGuidAnterior,
    xCritico := 1,
    sDescricao := 'Iniciado processo sem pesagem',
    sTag := 'IniSemPeso',
    iCamara := iCamara,
    stHoraAgora := stHoraAhora); // FB_SalvaEventoRelatorio

// NETWORK 10
fbSalvaEvento[10](
    sGuid := sGuidAnterior,
    xCritico := 1,
    sDescricao := 'Finalizado processo sem pesagem',
    sTag := 'FimSemPeso',
    iCamara := iCamara,
    stHoraAgora := stHoraAhora); // FB_SalvaEventoRelatorio
END_ACTION

ACTION fimAspersao:


IF xSalvaFimAspersao THEN
	
	FOR i:= 0 TO 50 DO
		saAux[i]:= '';
	END_FOR

	saAux[0] := ('UPDATE `geral`.`processos` SET `FimAspersao` = $'');
	saAux[1] := TO_STRING(stHoraAhora.wYear);
	saAux[2] := ('-');
	saAux[3] := (TO_STRING(stHoraAhora.wMonth));
	saAux[4] := ('-');
	saAux[5] := (TO_STRING(stHoraAhora.wDay));
	saAux[6] := (' ');
	saAux[7] := (TO_STRING(stHoraAhora.wHour));
	saAux[8] := (':');
	saAux[9] := (TO_STRING(stHoraAhora.wMinute));
	saAux[10] := (':');
	saAux[11] := (TO_STRING(stHoraAhora.wSecond));
	saAux[12] := ('$' WHERE (`Processo` = $'');
	saAux[13] := (sGuidAnterior);
	saAux[14] := ('$');');
	
	sCmd := F_ConcatArray1000(sArray:= saAux);
	
	aPara.eParaType := E_ExpParameterType.STRING_;
	aPara.nParaSize := SIZEOF(sAux);

	// call functionblock
	IF fbPLCDBaspersao.Execute(
		hDBID:= 1, 
		pExpression:= ADR(sCmd), 
		cbExpression:= SIZEOF(sCmd), 
		pData:= ADR(sAux), 
		cbData:= SIZEOF(sAux), 
		pParameter:= ADR(aPara), 
		cbParameter:= SIZEOF(aPara)) 
	THEN
		IF NOT fbPLCDBaspersao.bError THEN
			xSalvaFimAspersao := FALSE;
		END_IF
	END_IF
END_IF
END_ACTION

ACTION FimResfriamento:



//UPDATE `geral`.`processos` SET `InicioResfriamento` = '1', `NumeroCarcacas` = '1' WHERE (`Processo` = '{F4C353B8-2323-45D1-B9F0-8A1F447BE435}');


IF xSalvaFimResfriamento  THEN
	
	FOR i:= 0 TO 50 DO
		saAux[i]:= '';
	END_FOR
	
	saAux[0] := ('UPDATE `geral`.`processos` SET `FimResfriamento` = $'');
	saAux[2] := (TO_STRING(camara.en.stHoraAgora.wYear));
	saAux[3] := ('-');
	saAux[4] := (TO_STRING(camara.en.stHoraAgora.wMonth));
	saAux[5] := ('-');
	saAux[6] := (TO_STRING(camara.en.stHoraAgora.wDay));
	saAux[7] := (' ');
	saAux[8] := (TO_STRING(camara.en.stHoraAgora.wHour));
	saAux[9] := (':');
	saAux[10] := (TO_STRING(camara.en.stHoraAgora.wMinute));
	saAux[11] := (':');
	saAux[12] := (TO_STRING(camara.en.stHoraAgora.wSecond));
	saAux[13] := ('$', `NumeroCarcacas` = $'');
	saAux[14] := (TO_STRING(Camara.config.iCarcacasReal));
	saAux[15] := ('$' WHERE (`Processo` = $'');
	saAux[16] := (sGuidAnterior);
	saAux[17] := ('$');');
	
	sCmd := F_ConcatArray1000(sArray:= saAux);
	
	aPara.eParaType := E_ExpParameterType.STRING_;
	aPara.nParaSize := SIZEOF(sAux);

	// call functionblock
	IF fbPLCDBResfriamento.Execute(
		hDBID:= 1, 
		pExpression:= ADR(sCmd), 
		cbExpression:= SIZEOF(sCmd), 
		pData:= ADR(sAux), 
		cbData:= SIZEOF(sAux), 
		pParameter:= ADR(aPara), 
		cbParameter:= SIZEOF(aPara)) 
	THEN
		IF NOT fbPLCDBResfriamento.bError THEN
			xSalvaFimResfriamento := FALSE;
		END_IF
	END_IF
END_IF
END_ACTION

ACTION GeraRelatorio:

tonPodeGerarRelatorio(IN:= TRUE, PT:= T#2M, Q=> , ET=> );
IF NOT tonPodeGerarRelatorio.q THEN
	xGeraRelatorio := false;
END_IF


IF xGeraRelatorio AND tonPodeGerarRelatorio.q THEN
	
	FOR i:= 0 TO 50 DO
		saAux[i]:= '';
	END_FOR
	
	saAux[0]:= 'C:\TwinCAT\Asp.exe ';
	saAux[1]:= sGuidAnterior;
	saAux[2]:= ' ';
	saAux[3]:= Camara.config.sAbreviacaoUnidade;
	saAux[4]:= ' ';
	saAux[5]:= Camara.config.sIPFTP;
	
		
	sComando := F_ConcatArray1000(sArray:= saAux);
	
	
	fbProcessoEmail(
		NETID:= , 
		PATHSTR:= sComando, 
		DIRNAME:= , 
		COMNDLINE:= , 
		START:= xGeraRelatorio, 
		TMOUT:= , 
		BUSY=> , 
		ERR=> , 
		ERRID=> );
	
	IF NOT fbProcessoEmail.BUSY THEN
		xGeraRelatorio := FALSE;
		fbProcessoEmail(START:= FALSE);
	END_IF

END_IF
END_ACTION

ACTION InicioAspercao:


IF xSalvaInicioAspersao THEN
	
	Camara.sa.sHoraInicio :=  REPLACE(STR1:= TO_STRING(SYSTEMTIME_TO_DT(camara.en.stHoraAgora)), STR2:= '', L:= 15, P:=0);
	
	FOR i:= 0 TO 50 DO
		saAux[i]:= '';
	END_FOR

	saAux[0] := ('UPDATE `geral`.`processos` SET `InicioAspersao` = $'');
	saAux[1] := (TO_STRING(camara.en.stHoraAgora.wYear));
	saAux[2] := ('-');
	saAux[3] := (TO_STRING(camara.en.stHoraAgora.wMonth));
	saAux[4] := ('-');
	saAux[5] := (TO_STRING(camara.en.stHoraAgora.wDay));
	saAux[6] := (' ');
	saAux[7] := (TO_STRING(camara.en.stHoraAgora.wHour));
	saAux[8] := (':');
	saAux[9] := (TO_STRING(camara.en.stHoraAgora.wMinute));
	saAux[10] := (':');
	saAux[11] := (TO_STRING(camara.en.stHoraAgora.wSecond));
	saAux[12] := ('$' WHERE (`Processo` = $'');
	saAux[13] := (sGuidAnterior);
	saAux[14] := ('$');');
	
	sCmd := F_ConcatArray1000(sArray:= saAux);
	
	aPara.eParaType := E_ExpParameterType.STRING_;
	aPara.nParaSize := SIZEOF(sAux);

	// call functionblock
	IF fbPLCDBaspersao.Execute(
		hDBID:= 1, 
		pExpression:= ADR(sCmd), 
		cbExpression:= SIZEOF(sCmd), 
		pData:= ADR(sAux), 
		cbData:= SIZEOF(sAux), 
		pParameter:= ADR(aPara), 
		cbParameter:= SIZEOF(aPara)) 
	THEN
		IF NOT fbPLCDBaspersao.bError THEN
			xSalvaInicioAspersao := FALSE;
		END_IF
	END_IF
END_IF
END_ACTION

ACTION InicioResfriamento:



//UPDATE `geral`.`processos` SET `InicioResfriamento` = '1', `NumeroCarcacas` = '1' WHERE (`Processo` = '{F4C353B8-2323-45D1-B9F0-8A1F447BE435}');


IF xSalvaResfriamento THEN
	
	FOR i:= 0 TO 50 DO
		saAux[i]:= '';
	END_FOR
	
	saAux[0] := ('UPDATE `geral`.`processos` SET `InicioResfriamento` = $'');
	saAux[2] := (TO_STRING(camara.en.stHoraAgora.wYear));
	saAux[3] := ('-');
	saAux[4] := (TO_STRING(camara.en.stHoraAgora.wMonth));
	saAux[5] := ('-');
	saAux[6] := (TO_STRING(camara.en.stHoraAgora.wDay));
	saAux[7] := (' ');
	saAux[8] := (TO_STRING(camara.en.stHoraAgora.wHour));
	saAux[9] := (':');
	saAux[10] := (TO_STRING(camara.en.stHoraAgora.wMinute));
	saAux[11] := (':');
	saAux[12] := (TO_STRING(stHoraAhora.wSecond));
	saAux[13] := ('$', `NumeroCarcacas` = $'');
	saAux[14] := (TO_STRING(Camara.config.iCarcacasReal));
	saAux[15] := ('$' WHERE (`Processo` = $'');
	saAux[16] := (sGuidAnterior);
	saAux[17] := ('$');');
	
	sCmd := F_ConcatArray1000(sArray:= saAux);
	
	aPara.eParaType := E_ExpParameterType.STRING_;
	aPara.nParaSize := SIZEOF(sAux);

	// call functionblock
	IF fbPLCDBResfriamento.Execute(
		hDBID:= 1, 
		pExpression:= ADR(sCmd), 
		cbExpression:= SIZEOF(sCmd), 
		pData:= ADR(sAux), 
		cbData:= SIZEOF(sAux), 
		pParameter:= ADR(aPara), 
		cbParameter:= SIZEOF(aPara)) 
	THEN
		IF NOT fbPLCDBResfriamento.bError THEN
			xSalvaResfriamento := FALSE;
		END_IF
	END_IF
END_IF
END_ACTION

ACTION SalvaGrafico:



//INSERT INTO `geral`.`graficosprocesso` (`Processo`, `rTempTanque`, `rPressaoAnel`, `rUmidadeCamara`, `timestamp`) VALUES ('s', 's', 's', 's', 's');

tonAmostra(IN:= sGuidAtual <> '' AND xAmostra, PT:= T#5S, Q=> , ET=> );
IF tonAmostra.q THEN
	tonAmostra(IN:= FALSE);
	xSalvaGrafico := TRUE;
END_IF


IF xSalvaGrafico THEN
	
	FOR i:= 0 TO 50 DO
		saAux[i]:= '';
	END_FOR
	
	
	saAux[0]:= ('INSERT INTO `geral`.`graficosprocesso` (`Processo`, `rTempTanque`, `rPressao');
	saAux[1]:= ('Anel`, `rUmidadeCamara`, `rTemperaturaCamara`, `timestamp`) VALUES ($'');
	saAux[2]:= (sGuidAnterior);
	saAux[3]:= ('$', $'');
	saAux[4]:= (TO_STRING(F_RetiraCasa(Entrada:= Camara.en.rTempTanque, casa:=2)));
	saAux[5]:= ('$', $'');
	saAux[6]:= (TO_STRING(F_RetiraCasa(Entrada:= Camara.en.rPressaoAnel, casa:=2)));
	saAux[7]:= ('$', $'');
	saAux[8]:= (TO_STRING(F_RetiraCasa(Entrada:= Camara.en.rUmidadeCamara, casa:=2)));
	saAux[9]:= ('$', $'');
	saAux[10]:= (TO_STRING(F_RetiraCasa(Entrada:= Camara.en.rTempCamara, casa:=2)));
	saAux[11]:= ('$', $'');
	saAux[12]:= (TO_STRING(camara.en.stHoraAgora.wYear));
	saAux[13]:= ('-');
	saAux[14]:= (TO_STRING(camara.en.stHoraAgora.wMonth));
	saAux[15]:= ('-');
	saAux[16]:= (TO_STRING(camara.en.stHoraAgora.wDay));
	saAux[17]:= (' ');
	saAux[18]:= (TO_STRING(camara.en.stHoraAgora.wHour));
	saAux[19]:= (':');
	saAux[20]:= (TO_STRING(camara.en.stHoraAgora.wMinute));
	saAux[21]:= (':');
	saAux[22]:= (TO_STRING(camara.en.stHoraAgora.wSecond));
	saAux[23]:= ('$');');
	
	sCmd := F_ConcatArray1000(sArray:= saAux);
	
	aPara.eParaType := E_ExpParameterType.STRING_;
	aPara.nParaSize := SIZEOF(sAux);

	// call functionblock
	IF fbPLCDBCmd.Execute(
		hDBID:= 1, 
		pExpression:= ADR(sCmd), 
		cbExpression:= SIZEOF(sCmd), 
		pData:= ADR(sAux), 
		cbData:= SIZEOF(sAux), 
		pParameter:= ADR(aPara), 
		cbParameter:= SIZEOF(aPara)) 
	THEN
		xSalvaGrafico := FALSE;
	END_IF
END_IF
END_ACTION

ACTION SalvaProtocolo:

IF xSalvaProtocolo THEN
		
	FOR i:= 0 TO 50 DO
		saAux[i]:= '';
	END_FOR

	//UPDATE `geral`.`processos` SET `sProtocolo` = 'aaaaaaa' WHERE (`Processo` = '{008089BB-BE64-417E-ABDE-888FE5FB9663}');

	saAux[0] := ('UPDATE `geral`.`processos` SET `sProtocolo` = $'');
	saAux[1] := (Camara.config.stProtocolos[Camara.config.iProtocoloEscolhido].DB.Nome);
	saAux[2] := ('$' WHERE (`Processo` = $'');
	saAux[3] := (sGuidAnterior);
	saAux[4] := ('$');');
	
	sCmd := F_ConcatArray1000(sArray:= saAux);
	
	aPara.eParaType := E_ExpParameterType.STRING_;
	aPara.nParaSize := SIZEOF(sAux);

	// call functionblock
	IF fbPLCDProtocolo.Execute(
		hDBID:= 1, 
		pExpression:= ADR(sCmd), 
		cbExpression:= SIZEOF(sCmd), 
		pData:= ADR(sAux), 
		cbData:= SIZEOF(sAux), 
		pParameter:= ADR(aPara), 
		cbParameter:= SIZEOF(aPara)) 
	THEN
		IF NOT fbPLCDProtocolo.bError THEN
			xSalvaProtocolo := FALSE;
		END_IF
	END_IF
END_IF
END_ACTION

ACTION AjustaEntrada:



IF Camara.config.iCamara <> CamaraAnterior.config.iCamara THEN
	iCamara := Camara.config.iCamara;
END_IF
IF Camara.config.iCamara <> iCamara THEN
	Camara.config.iCamara := iCamara;
END_IF


IF Camara.config.sNome <> CamaraAnterior.config.sNome THEN
	sNome := Camara.config.sNome;
END_IF
IF Camara.config.sNome <> sNome THEN
	Camara.config.sNome := sNome;
END_IF


IF Camara.en.sGuidAtual <> CamaraAnterior.en.sGuidAtual THEN
	sGuidAtual := Camara.en.sGuidAtual;
END_IF
IF Camara.en.sGuidAtual <> sGuidAtual THEN
	Camara.en.sGuidAtual := sGuidAtual;
END_IF


IF Camara.config.sValvulas <> CamaraAnterior.config.sValvulas THEN
	sValvulas := Camara.config.sValvulas;
	F_StringSeparadorFBGrupos(sStr:= sValvulas, ListaINT:=iValvulas);
END_IF
IF Camara.config.sValvulas <> sValvulas THEN
	Camara.config.sValvulas := sValvulas;
	F_StringSeparadorFBGrupos(sStr:= sValvulas, ListaINT:=iValvulas);
END_IF


IF Camara.status.xCamaraTempOK <> CamaraAnterior.status.xCamaraTempOK THEN
	xCamaraTempOK := Camara.status.xCamaraTempOK;
END_IF
IF Camara.status.xCamaraTempOK <> xCamaraTempOK THEN
	Camara.status.xCamaraTempOK := xCamaraTempOK;
END_IF

IF Camara.status.xCamaraUmidOK <> CamaraAnterior.status.xCamaraUmidOK THEN
	xCamaraUmidOK := Camara.status.xCamaraUmidOK;
END_IF
IF Camara.status.xCamaraUmidOK <> xCamaraUmidOK THEN
	Camara.status.xCamaraUmidOK := xCamaraUmidOK;
END_IF

IF Camara.status.xAnelPressOK <> CamaraAnterior.status.xAnelPressOK THEN
	xAnelPressOK := Camara.status.xAnelPressOK;
END_IF
IF Camara.status.xAnelPressOK <> xAnelPressOK THEN
	Camara.status.xAnelPressOK := xAnelPressOK;
END_IF

IF Camara.status.xTanqueTempOK <> CamaraAnterior.status.xTanqueTempOK THEN
	xTanqueTempOK := Camara.status.xTanqueTempOK;
END_IF
IF Camara.status.xTanqueTempOK <> xTanqueTempOK THEN
	Camara.status.xTanqueTempOK := xTanqueTempOK;
END_IF

IF Camara.en.xFinalizaValvulasDaCamara <> CamaraAnterior.en.xFinalizaValvulasDaCamara THEN
	xFinalizaValvulasDaCamara := Camara.en.xFinalizaValvulasDaCamara;
END_IF
IF Camara.en.xFinalizaValvulasDaCamara <> xFinalizaValvulasDaCamara THEN
	Camara.en.xFinalizaValvulasDaCamara := xFinalizaValvulasDaCamara;
END_IF

//Quantidade minima de carcaças a amostrar
IF Camara.config.iCarcacasAmostra < 20 THEN
	Camara.config.iCarcacasAmostra := 20;
END_IF



CamaraAnterior := Camara;
END_ACTION

ACTION AjustaSaida:




Camara.status.sStatus := sStatus;
Camara.status.iStatus := iStatus;
Camara.status.xTerminouAspercao := xTerminouAspercao;
Camara.sa.iQuantidadeDeCluster := iQuantidadeDeCluster;

Camara.status.sNomeProtocoloAtivo := Camara.config.stProtocolos[Camara.config.iProtocoloEscolhido].DB.Nome;



Camara.sa.iValvulaMestraMestra := iValvulaMestraMestra;
END_ACTION

ACTION ControleLed:


ton10s(IN:=TRUE, PT:= T#10S, Q=> , ET=> );
IF ton10s.q THEN
	ton10s(IN:=TRUE);
	x10s := NOT x10s;
END_IF

ton2s(IN:=TRUE, PT:= T#2S, Q=> , ET=> );
IF ton2s.q THEN
	ton2s(IN:=TRUE);
	x2s := NOT x2s;
END_IF

ton500ms(IN:=TRUE, PT:= T#500MS, Q=> , ET=> );
IF ton500ms.q THEN
	ton500ms(IN:=TRUE);
	x500ms := NOT x500ms;
END_IF


IF sGuidAtual = '' THEN
	Camara.sa.xLed := FALSE;	
END_IF

IF sGuidAtual <> '' AND NOT xIniciouAspercao THEN
	Camara.sa.xLed := x2s;
END_IF

IF sGuidAtual <> '' AND xIniciouAspercao THEN
	Camara.sa.xLed := TRUE;
END_IF

IF sGuidAtual <> '' AND xTerminouAspercao THEN
	Camara.sa.xLed := x10s AND x2s;
END_IF



IF Camara.en.xLedManual THEN
	Camara.sa.xLed := Camara.en.xSinalManuLed;
END_IF
END_ACTION

ACTION InicioPelaCamara:



CASE iMaquinaIniciaSemPeso OF
	0://Esperando ter que criar um guid e salvar no banco
		IF (Camara.en.xIniciaCamaraSupervisorio OR Camara.en.xIniciaCamaraIHM) AND sGuidAtual = '' THEN
			iMaquinaIniciaSemPeso := 1;
			Camara.en.xIniciaCamaraSupervisorio := FALSE;
			Camara.en.xIniciaCamaraIHM := FALSE;
		END_IF
		
	1: // cria o guid
	
		fbCriaGUID(
			bExecute:= TRUE,  
			sNetId:= '', 
			tTimeout:= T#5S, 
			pGuidBuffer:= ADR(guidCriado), 
			nGuidBufferSize:= SIZEOF(guidCriado), 
			bBusy=> , 
			bError=> , 
			nErrorId=> );
			
		IF NOT fbCriaGUID.bBusy THEN
			fbCriaGUID(bExecute:= FALSE);
			sGuidAtual := GUID_TO_REGSTRING(guidCriado);
			iMaquinaIniciaSemPeso := 2;
		END_IF
		
	2://salva no banco o role
		FOR i:= 0 TO 50 DO
			saAux[i]:= '';
		END_FOR
	
		saAux[0] := ('INSERT INTO `geral`.`processos` (`Processo`');
		saAux[1] := (', `Camara`, `Status`,`InicioResfriamento`, `Timestamp`) VALUES ($'');
		saAux[2] := sGuidAtual;
		saAux[3] := '$', $'';
		saAux[4] := TO_STRING(Camara.config.iCamara);
		saAux[5] := '$', $'';
		saAux[6] := 'Esperando aspersao';
		saAux[7] := '$', $'';
		saAux[8] := TO_STRING(stHoraAhora.wYear);
		saAux[9] := ('-');
		saAux[10] := (TO_STRING(stHoraAhora.wMonth));
		saAux[11] := ('-');
		saAux[12] := (TO_STRING(stHoraAhora.wDay));
		saAux[13] := (' ');
		saAux[14] := (TO_STRING(stHoraAhora.wHour));
		saAux[15] := (':');
		saAux[16] := (TO_STRING(stHoraAhora.wMinute));
		saAux[17] := (':');
		saAux[18] := (TO_STRING(stHoraAhora.wSecond));
		saAux[19] := '$', $'';
		saAux[20] := TO_STRING(stHoraAhora.wYear);
		saAux[21] := ('-');
		saAux[22] := (TO_STRING(stHoraAhora.wMonth));
		saAux[23] := ('-');
		saAux[24] := (TO_STRING(stHoraAhora.wDay));
		saAux[25] := (' ');
		saAux[26] := (TO_STRING(stHoraAhora.wHour));
		saAux[27] := (':');
		saAux[28] := (TO_STRING(stHoraAhora.wMinute));
		saAux[29] := (':');
		saAux[30] := (TO_STRING(stHoraAhora.wSecond));
		saAux[31] := ('$');');
		
		sCmd := F_ConcatArray1000(sArray:= saAux);
		
		aPara.eParaType := E_ExpParameterType.STRING_;
		aPara.nParaSize := SIZEOF(sAux);
	
		// call functionblock
		IF fbDBInicioProcesso.Execute(
			hDBID:= 1, 
			pExpression:= ADR(sCmd), 
			cbExpression:= SIZEOF(sCmd), 
			pData:= ADR(sAux), 
			cbData:= SIZEOF(sAux), 
			pParameter:= ADR(aPara), 
			cbParameter:= SIZEOF(aPara)) 
		THEN
			IF NOT fbDBInicioProcesso.bError THEN
				xSalvaIniSemPeso := TRUE;
				iMaquinaIniciaSemPeso := 0;
			END_IF
		END_IF
END_CASE
END_ACTION

ACTION Status:



IF sGuidAtual = '' THEN
	sStatus := 'StandBy';
	iStatus := 1;
ELSE
	
	IF Camara.Status.xPegandoPesosQuentes THEN
		sStatus := 'Aquisitando pesos quentes';
		iStatus := 8;
	END_IF
	
	IF NOT xIniciouAspercao AND NOT Camara.Status.xPegandoPesosQuentes THEN
		sStatus := 'Esperando o incio da aspersão';
		iStatus := 2;
	END_IF
	
	IF NOT xTerminouAspercao AND xIniciouAspercao THEN
		sStatus := 'Esperando o fim da aspersão';
		iStatus := 3;
	END_IF
	
	IF xTerminouAspercao THEN
		sStatus := 'Aspersão finalizada';
		iStatus	 := 4;
	END_IF
	
	
	IF Camara.Status.xPegandoPesosFrios THEN
		sStatus := 'Aquisitando pesos frios';
		iStatus := 9;
	END_IF
	
	//Abaixo os prioritarios sobre esses de cima
	
	IF Camara.Status.xPeloMenos1CanceladaOutrasAguradando OR Camara.Status.xTodasValvulasCanceladas THEN
		iStatus	 := 6;
	END_IF
	
	IF Camara.Status.xAlgumaValvulaEmManual THEN
		iStatus	 := 7;
	END_IF
	
	IF (NOT xCamaraTempOK OR NOT xCamaraUmidOK OR NOT xAnelPressOK OR NOT xTanqueTempOK) AND NOT xTerminouAspercao THEN	
		iStatus	 := 5;		
	END_IF
END_IF



//Tem alguma Valvula em manual
Camara.Status.xAlgumaValvulaEmManual := FALSE;
FOR i := 0 TO 500 DO
	IF iValvulas[i] = 0 THEN
		EXIT;
	ELSE
		IF NOT stControleValvulas[iValvulas[i]].EN.stValvula.en.xAutomaticoManual THEN
			Camara.Status.xAlgumaValvulaEmManual := TRUE;	
		END_IF
	END_IF
END_FOR



